// TIA Portal project "ProgettoTisc_Gruppo19" (V17)

(* hardware
DEVICE "S7-1200 station_1"  S7-1200 Station
   slot 0: "Rack_0"  S7-1200 Rack  Rack  V1.0
   slot 1: "PLC_1"  CPU 1211C DC/DC/DC  6ES7 211-1AE40-0XB0  V4.5
DEVICE "HMI_1"  KTP900 Basic PN
   slot 0: "HMI_1"  KTP900 Basic PN  6AV2 123-2JB03-0AX0  17.0.0.0
   slot 1: "HMI_RT_1"  KTP900 Basic PN  6AV2 123-2JB03-0AX0  17.0.0.0
   slot 5: "HMI_1.IE_CP_1"  PROFINET Interface  17.0.0.0
      slot 1: "PROFINET Interface_1"  PROFINET Interface
         slot 1: "Port_1"  Port
*)

// ===== PLC "PLC_1"  CPU 1211C DC/DC/DC =====

VAR_GLOBAL   // PLC tag table "Default tag table"
   "S1" AT %I10.0 : Bool;
   "Sh1" AT %I10.1 : Bool;
   "detected" AT %I10.2 : Bool;
   "X_position" AT %ID32 : Real;
   "Y_position" AT %ID36 : Real;
   "Z_position" AT %ID40 : Real;
   "S2" AT %I10.3 : Bool;
   "Sn1" AT %I10.4 : Bool;
   "S_dx" AT %I10.5 : Bool;
   "Sn_dx" AT %I10.6 : Bool;
   "Sc_value_dx" AT %ID44 : DInt;
   "exit_limit_dx" AT %I10.7 : Bool;
   "enter_limit_dx" AT %I11.0 : Bool;
   "position_dx" AT %ID48 : Real;
   "S_sx" AT %I11.1 : Bool;
   "Sn_sx" AT %I11.2 : Bool;
   "Sc_value_sx" AT %ID52 : DInt;
   "exit_limit_sx" AT %I11.3 : Bool;
   "enter_limit_sx" AT %I11.4 : Bool;
   "position_sx" AT %ID56 : Real;
   "motor1" AT %Q0.0 : Bool;
   "X_setpoint" AT %QD30 : Real;
   "Y_setpoint" AT %QD34 : Real;
   "Z_setpoint" AT %QD38 : Real;
   "grab" AT %Q0.1 : Bool;
   "motor2" AT %Q0.2 : Bool;
   "move" AT %Q0.3 : Bool;
   "move_right" AT %Q0.4 : Bool;
   "move_left" AT %Q0.5 : Bool;
   "motor_dx" AT %Q0.6 : Bool;
   "roll_dx" AT %Q0.7 : Bool;
   "motor1_dx" AT %Q1.0 : Bool;
   "motor2_dx" AT %Q1.1 : Bool;
   "motor3_dx" AT %Q1.2 : Bool;
   "setpoint_dx" AT %QD42 : Real;
   "motor_sx" AT %Q1.3 : Bool;
   "roll_sx" AT %Q1.4 : Bool;
   "motor1_sx" AT %Q1.5 : Bool;
   "motor2_sx" AT %Q1.6 : Bool;
   "motor3_sx" AT %Q1.7 : Bool;
   "setpoint_sx" AT %QD46 : Real;
   "Emitter_pallet" AT %Q2.0 : Bool;
   "Emitter_basi" AT %Q2.1 : Bool;
   "Impianto_attivo" AT %M0.0 : Bool;
   "Cmd_start" AT %M0.1 : Bool;
   "Cmd_stop" AT %M0.2 : Bool;
   "Pezzi_totali" AT %MW10 : Int;
   "Pezzi_blu" AT %MW12 : Int;
   "Pezzi_verdi" AT %MW14 : Int;
   "Pezzi_grigi" AT %MW16 : Int;
   "Allarme" AT %M0.3 : Bool;
   "Reset" AT %M0.4 : Bool;
   "Sospendi" AT %M0.5 : Bool;
   "Allarme_colore_dx" AT %M0.6 : Bool;
   "Allarme_colore_sx" AT %M0.7 : Bool;
   "Allarme_sh" AT %M1.0 : Bool;
   "Sirena_allarmi" AT %Q2.2 : Bool;
   "Flash_Sh" AT %Q2.3 : Bool;
   "Flash_dx" AT %Q2.4 : Bool;
   "Flash_sx" AT %Q2.5 : Bool;
   "Allarme_sh_int" AT %MW20 : Int;
   "Allarme_colore_dx_int" AT %MW22 : Int;
   "Allarme_colore_sx_int" AT %MW24 : Int;
   "Attesa_sh" AT %M1.1 : Bool;
   "Attesa_controllo_colore_dx" AT %M1.2 : Bool;
   "Attesa_controllo_colore_sx" AT %M1.3 : Bool;
END_VAR

DATA_BLOCK "Nastro_di_produzione_DB"   // DB1
{ S7_Optimized_Access := 'TRUE' }
VERSION : 0.1
// stored: InstanceOfName Nastro_di_produzione
"Nastro_di_produzione"
BEGIN
END_DATA_BLOCK

DATA_BLOCK "Pick-place_DB"   // DB2
{ S7_Optimized_Access := 'TRUE' }
VERSION : 0.1
// stored: InstanceOfName Pick-place
"Pick-place"
BEGIN
END_DATA_BLOCK

DATA_BLOCK "Nastro_DB"   // DB3
{ S7_Optimized_Access := 'TRUE' }
VERSION : 0.1
// stored: InstanceOfName Nastro
"Nastro"
BEGIN
END_DATA_BLOCK

DATA_BLOCK "Transfer_DB"   // DB4
{ S7_Optimized_Access := 'TRUE' }
VERSION : 0.1
// stored: InstanceOfName Transfer
"Transfer"
BEGIN
END_DATA_BLOCK

DATA_BLOCK "Nastro_di_smistamento_dx_DB"   // DB5
{ S7_Optimized_Access := 'TRUE' }
VERSION : 0.1
// stored: InstanceOfName Nastro_di_smistamento
"Nastro_di_smistamento"
BEGIN
END_DATA_BLOCK

DATA_BLOCK "Elevator_dx_DB"   // DB6
{ S7_Optimized_Access := 'TRUE' }
VERSION : 0.1
// stored: InstanceOfName Elevator
"Elevator"
BEGIN
END_DATA_BLOCK

DATA_BLOCK "Nastro_di_smistamento_sx_DB"   // DB7
{ S7_Optimized_Access := 'TRUE' }
VERSION : 0.1
// stored: InstanceOfName Nastro_di_smistamento
"Nastro_di_smistamento"
BEGIN
END_DATA_BLOCK

DATA_BLOCK "Elevator_sx_DB"   // DB8
{ S7_Optimized_Access := 'TRUE' }
VERSION : 0.1
// stored: InstanceOfName Elevator
"Elevator"
BEGIN
END_DATA_BLOCK

DATA_BLOCK "Supervisore_DB"   // DB12
{ S7_Optimized_Access := 'TRUE' }
VERSION : 0.1
// stored: InstanceOfName Supervisore
"Supervisore"
BEGIN
END_DATA_BLOCK

// folder: System blocks/Program resources

DATA_BLOCK "TON_Allarme_Sh_DB"   // DB13
{ S7_Optimized_Access := 'TRUE' }
AUTHOR : Simatic
FAMILY : IEC
NAME : IEC_TMR
VERSION : 1.0
// stored: InstanceOfName IEC_TIMER
"IEC_TIMER"
BEGIN
END_DATA_BLOCK

DATA_BLOCK "TON_Allarme_dx"   // DB14
{ S7_Optimized_Access := 'TRUE' }
AUTHOR : Simatic
FAMILY : IEC
NAME : IEC_TMR
VERSION : 1.0
// stored: InstanceOfName IEC_TIMER
"IEC_TIMER"
BEGIN
END_DATA_BLOCK

DATA_BLOCK "TON_Allarme_sx"   // DB15
{ S7_Optimized_Access := 'TRUE' }
AUTHOR : Simatic
FAMILY : IEC
NAME : IEC_TMR
VERSION : 1.0
// stored: InstanceOfName IEC_TIMER
"IEC_TIMER"
BEGIN
END_DATA_BLOCK

// folder: (top level)

FUNCTION_BLOCK "Nastro_di_produzione"   // FB1, LAD
{ S7_Optimized_Access := 'TRUE' }
VERSION : 0.1
   VAR_INPUT
      S : Bool;
      work_finished : Bool;
      Sh : Bool;
      p_dopo : Bool;
      Sospendi : Bool;
      Forza : Bool;
   END_VAR
   VAR_OUTPUT
      motor : Bool;
      work : Bool;
   END_VAR
   VAR
      p1 : Bool;
      p2 : Bool;
      p3 : Bool;
      p4 : Bool;
      p5 : Bool;
      t1 : Bool;
      t2 : Bool;
      t3 : Bool;
      t4 : Bool;
      t5 : Bool;
      R_TRIG_S : R_TRIG;
      R_TRIG_Sh : R_TRIG;
      F_TRIG_S : R_TRIG;
      INIZ : Bool;
   END_VAR
   VAR_TEMP   // added for the SCL form of the ladder/FBD networks
      _w1 : Bool;
   END_VAR
BEGIN

REGION Network 1: Inizializzazione
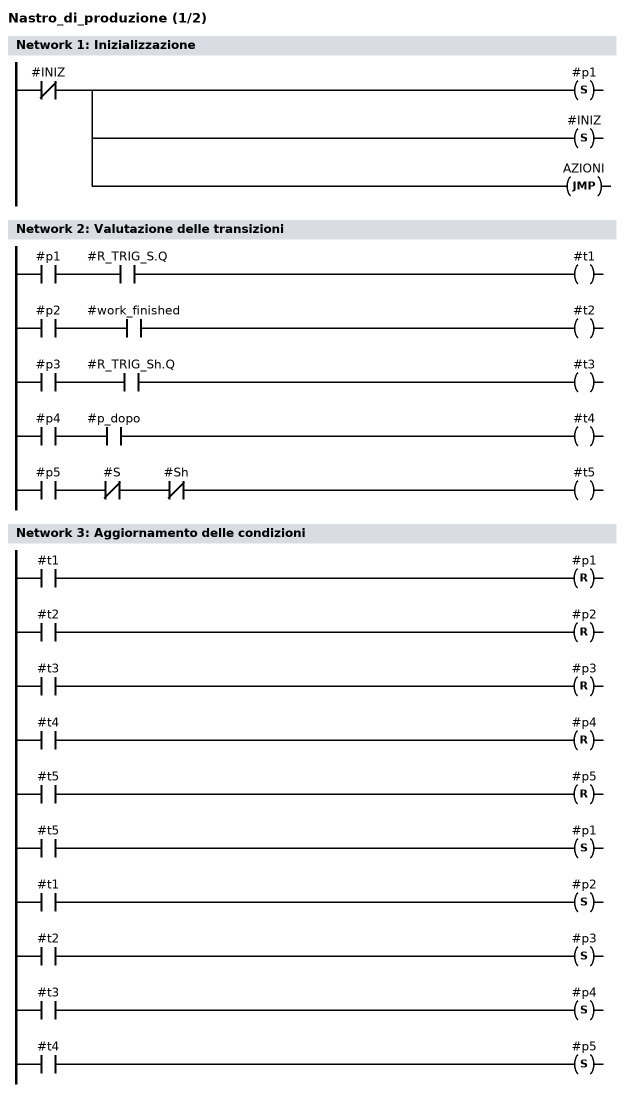
   RUNG wire#powerrail
      I_Contact( #INIZ )
      wire#w1
      S_Coil( #p1 )
   END_RUNG
   RUNG wire#w1
      S_Coil( #INIZ )
   END_RUNG
   RUNG wire#w1
      JumpCoil( AZIONI )
   END_RUNG
   // the same network as SCL:
   IF NOT #INIZ THEN #p1 := TRUE; END_IF;
   #_w1 := NOT #INIZ;
   IF #_w1 THEN
       #INIZ := TRUE;
       GOTO AZIONI;
   END_IF;
END_REGION

REGION Network 2: Valutazione delle transizioni
   RUNG wire#powerrail
      Contact( #p1 )
      Contact( #R_TRIG_S.Q )
      Coil( #t1 )
   END_RUNG
   RUNG wire#powerrail
      Contact( #p2 )
      Contact( #work_finished )
      Coil( #t2 )
   END_RUNG
   RUNG wire#powerrail
      Contact( #p3 )
      Contact( #R_TRIG_Sh.Q )
      Coil( #t3 )
   END_RUNG
   RUNG wire#powerrail
      Contact( #p4 )
      Contact( #p_dopo )
      Coil( #t4 )
   END_RUNG
   RUNG wire#powerrail
      Contact( #p5 )
      I_Contact( #S )
      I_Contact( #Sh )
      Coil( #t5 )
   END_RUNG
   // the same network as SCL:
   #t1 := #p1 AND #R_TRIG_S.Q;
   #t2 := #p2 AND #work_finished;
   #t3 := #p3 AND #R_TRIG_Sh.Q;
   #t4 := #p4 AND #p_dopo;
   #t5 := #p5 AND NOT #S AND NOT #Sh;
END_REGION

REGION Network 3: Aggiornamento delle condizioni
   RUNG wire#powerrail
      Contact( #t1 )
      R_Coil( #p1 )
   END_RUNG
   RUNG wire#powerrail
      Contact( #t2 )
      R_Coil( #p2 )
   END_RUNG
   RUNG wire#powerrail
      Contact( #t3 )
      R_Coil( #p3 )
   END_RUNG
   RUNG wire#powerrail
      Contact( #t4 )
      R_Coil( #p4 )
   END_RUNG
   RUNG wire#powerrail
      Contact( #t5 )
      R_Coil( #p5 )
   END_RUNG
   RUNG wire#powerrail
      Contact( #t5 )
      S_Coil( #p1 )
   END_RUNG
   RUNG wire#powerrail
      Contact( #t1 )
      S_Coil( #p2 )
   END_RUNG
   RUNG wire#powerrail
      Contact( #t2 )
      S_Coil( #p3 )
   END_RUNG
   RUNG wire#powerrail
      Contact( #t3 )
      S_Coil( #p4 )
   END_RUNG
   RUNG wire#powerrail
      Contact( #t4 )
      S_Coil( #p5 )
   END_RUNG
   // the same network as SCL:
   IF #t1 THEN #p1 := FALSE; END_IF;
   IF #t2 THEN #p2 := FALSE; END_IF;
   IF #t3 THEN #p3 := FALSE; END_IF;
   IF #t4 THEN #p4 := FALSE; END_IF;
   IF #t5 THEN
       #p5 := FALSE;
       #p1 := TRUE;
   END_IF;
   IF #t1 THEN #p2 := TRUE; END_IF;
   IF #t2 THEN #p3 := TRUE; END_IF;
   IF #t3 THEN #p4 := TRUE; END_IF;
   IF #t4 THEN #p5 := TRUE; END_IF;
END_REGION

REGION Network 4: Macroazioni di sospensione e forzatura alla fase 1 e sezione di esecuzione delle azioni
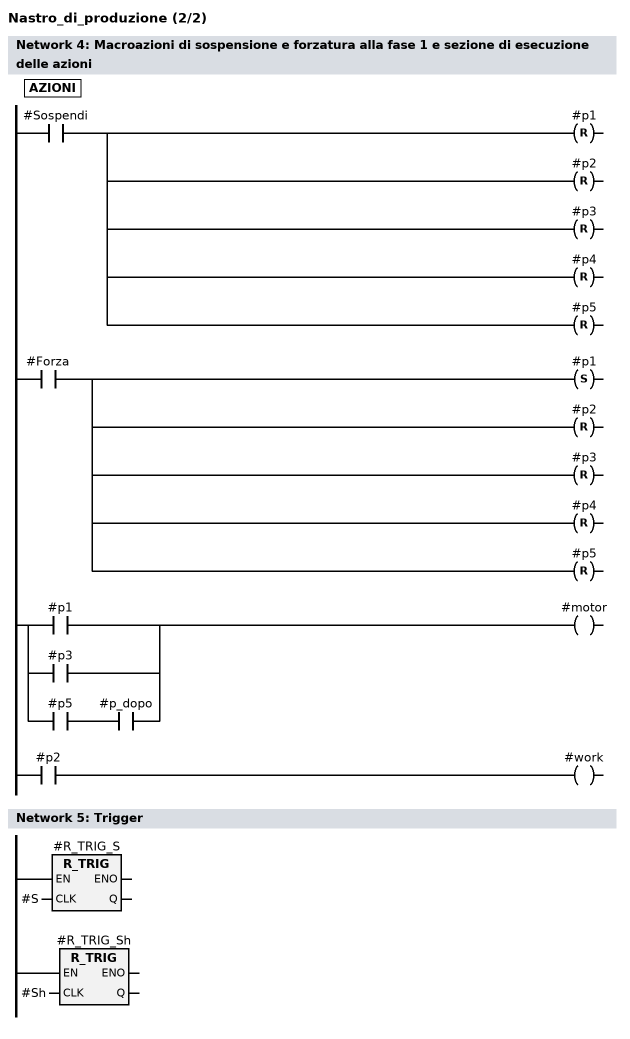
   Label( AZIONI )
   RUNG wire#powerrail
      Contact( #Sospendi )
      wire#w1
      R_Coil( #p1 )
   END_RUNG
   RUNG wire#w1
      R_Coil( #p2 )
   END_RUNG
   RUNG wire#w1
      R_Coil( #p3 )
   END_RUNG
   RUNG wire#w1
      R_Coil( #p4 )
   END_RUNG
   RUNG wire#w1
      R_Coil( #p5 )
   END_RUNG
   RUNG wire#powerrail
      Contact( #Forza )
      wire#w2
      S_Coil( #p1 )
   END_RUNG
   RUNG wire#w2
      R_Coil( #p2 )
   END_RUNG
   RUNG wire#w2
      R_Coil( #p3 )
   END_RUNG
   RUNG wire#w2
      R_Coil( #p4 )
   END_RUNG
   RUNG wire#w2
      R_Coil( #p5 )
   END_RUNG
   RUNG wire#powerrail
      Contact( #p1 )
      wire#w3
      Coil( #motor )
   END_RUNG
   RUNG wire#powerrail
      Contact( #p3 )
   END_RUNG wire#w3
   RUNG wire#powerrail
      Contact( #p5 )
      Contact( #p_dopo )
   END_RUNG wire#w3
   RUNG wire#powerrail
      Contact( #p2 )
      Coil( #work )
   END_RUNG
   // the same network as SCL:
   AZIONI:
   IF #Sospendi THEN
       #p1 := FALSE;
       #p2 := FALSE;
       #p3 := FALSE;
       #p4 := FALSE;
       #p5 := FALSE;
   END_IF;
   IF #Forza THEN
       #p1 := TRUE;
       #p2 := FALSE;
       #p3 := FALSE;
       #p4 := FALSE;
       #p5 := FALSE;
   END_IF;
   #motor := #p1 OR #p3 OR (#p5 AND #p_dopo);
   #work := #p2;
END_REGION

REGION Network 5: Trigger
   #R_TRIG_S(CLK := #S);   // R_TRIG
   #R_TRIG_Sh(CLK := #Sh);   // R_TRIG
END_REGION
END_FUNCTION_BLOCK

FUNCTION_BLOCK "Nastro"   // FB2, LAD
{ S7_Optimized_Access := 'TRUE' }
VERSION : 0.1
   VAR_INPUT
      S : Bool;
      p_dopo : Bool;
      Sospendi : Bool;
      Forza : Bool;
   END_VAR
   VAR_OUTPUT
      Motor : Bool;
      Pronto_ricevere : Bool;
      transfer : Bool;
   END_VAR
   VAR
      p1 : Bool;
      p2 : Bool;
      p3 : Bool;
      t1 : Bool;
      t2 : Bool;
      t3 : Bool;
      R_TRIG_S : R_TRIG;
      F_TRIG_S : F_TRIG;
      INIZ : Bool;
   END_VAR
   VAR_TEMP   // added for the SCL form of the ladder/FBD networks
      _w1 : Bool;
   END_VAR
BEGIN

REGION Network 1: Inizializzazione
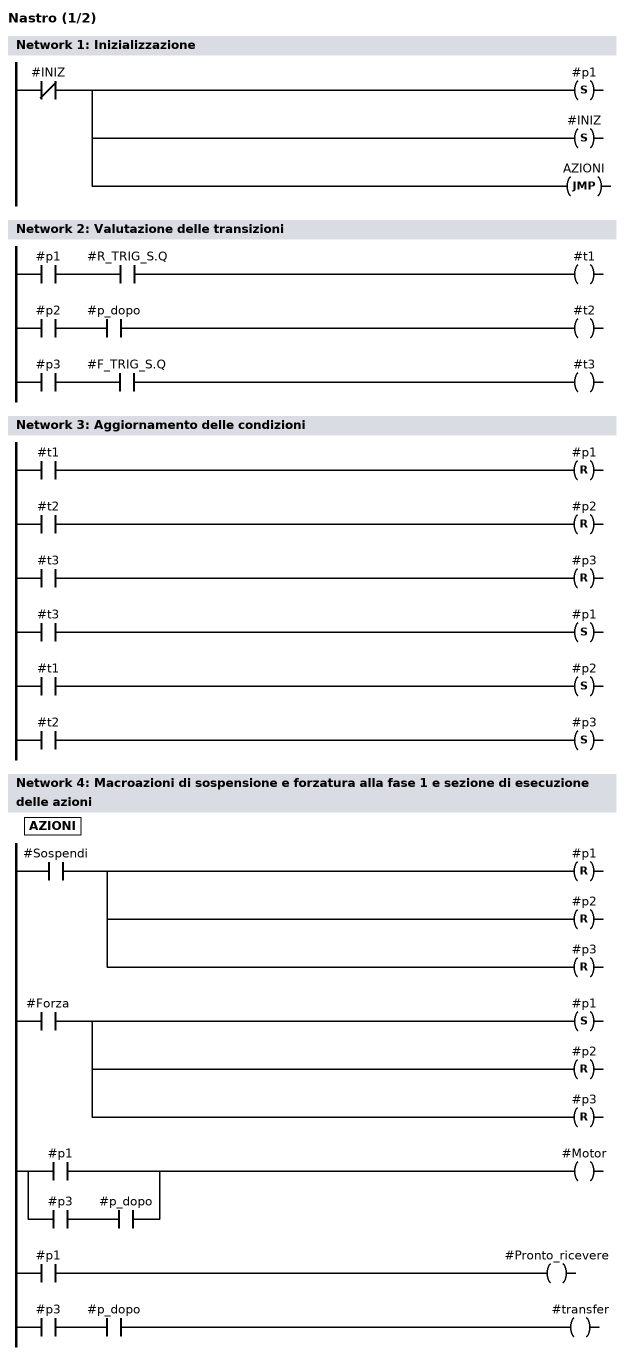
   RUNG wire#powerrail
      I_Contact( #INIZ )
      wire#w1
      S_Coil( #p1 )
   END_RUNG
   RUNG wire#w1
      S_Coil( #INIZ )
   END_RUNG
   RUNG wire#w1
      JumpCoil( AZIONI )
   END_RUNG
   // the same network as SCL:
   IF NOT #INIZ THEN #p1 := TRUE; END_IF;
   #_w1 := NOT #INIZ;
   IF #_w1 THEN
       #INIZ := TRUE;
       GOTO AZIONI;
   END_IF;
END_REGION

REGION Network 2: Valutazione delle transizioni
   RUNG wire#powerrail
      Contact( #p1 )
      Contact( #R_TRIG_S.Q )
      Coil( #t1 )
   END_RUNG
   RUNG wire#powerrail
      Contact( #p2 )
      Contact( #p_dopo )
      Coil( #t2 )
   END_RUNG
   RUNG wire#powerrail
      Contact( #p3 )
      Contact( #F_TRIG_S.Q )
      Coil( #t3 )
   END_RUNG
   // the same network as SCL:
   #t1 := #p1 AND #R_TRIG_S.Q;
   #t2 := #p2 AND #p_dopo;
   #t3 := #p3 AND #F_TRIG_S.Q;
END_REGION

REGION Network 3: Aggiornamento delle condizioni
   RUNG wire#powerrail
      Contact( #t1 )
      R_Coil( #p1 )
   END_RUNG
   RUNG wire#powerrail
      Contact( #t2 )
      R_Coil( #p2 )
   END_RUNG
   RUNG wire#powerrail
      Contact( #t3 )
      R_Coil( #p3 )
   END_RUNG
   RUNG wire#powerrail
      Contact( #t3 )
      S_Coil( #p1 )
   END_RUNG
   RUNG wire#powerrail
      Contact( #t1 )
      S_Coil( #p2 )
   END_RUNG
   RUNG wire#powerrail
      Contact( #t2 )
      S_Coil( #p3 )
   END_RUNG
   // the same network as SCL:
   IF #t1 THEN #p1 := FALSE; END_IF;
   IF #t2 THEN #p2 := FALSE; END_IF;
   IF #t3 THEN
       #p3 := FALSE;
       #p1 := TRUE;
   END_IF;
   IF #t1 THEN #p2 := TRUE; END_IF;
   IF #t2 THEN #p3 := TRUE; END_IF;
END_REGION

REGION Network 4: Macroazioni di sospensione e forzatura alla fase 1 e sezione di esecuzione delle azioni
   Label( AZIONI )
   RUNG wire#powerrail
      Contact( #Sospendi )
      wire#w1
      R_Coil( #p1 )
   END_RUNG
   RUNG wire#w1
      R_Coil( #p2 )
   END_RUNG
   RUNG wire#w1
      R_Coil( #p3 )
   END_RUNG
   RUNG wire#powerrail
      Contact( #Forza )
      wire#w2
      S_Coil( #p1 )
   END_RUNG
   RUNG wire#w2
      R_Coil( #p2 )
   END_RUNG
   RUNG wire#w2
      R_Coil( #p3 )
   END_RUNG
   RUNG wire#powerrail
      Contact( #p1 )
      wire#w3
      Coil( #Motor )
   END_RUNG
   RUNG wire#powerrail
      Contact( #p3 )
      Contact( #p_dopo )
   END_RUNG wire#w3
   RUNG wire#powerrail
      Contact( #p1 )
      Coil( #Pronto_ricevere )
   END_RUNG
   RUNG wire#powerrail
      Contact( #p3 )
      Contact( #p_dopo )
      Coil( #transfer )
   END_RUNG
   // the same network as SCL:
   AZIONI:
   IF #Sospendi THEN
       #p1 := FALSE;
       #p2 := FALSE;
       #p3 := FALSE;
   END_IF;
   IF #Forza THEN
       #p1 := TRUE;
       #p2 := FALSE;
       #p3 := FALSE;
   END_IF;
   #Motor := #p1 OR (#p3 AND #p_dopo);
   #Pronto_ricevere := #p1;
   #transfer := #p3 AND #p_dopo;
END_REGION

REGION Network 5: Trigger
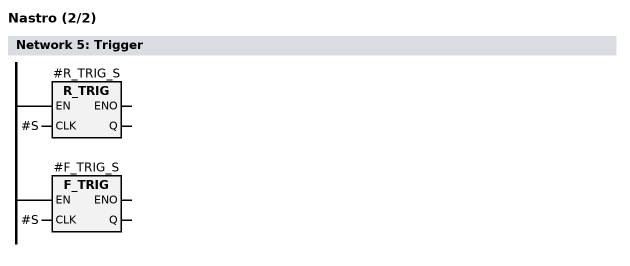
   #R_TRIG_S(CLK := #S);   // R_TRIG
   #F_TRIG_S(CLK := #S);   // F_TRIG
END_REGION
END_FUNCTION_BLOCK

FUNCTION_BLOCK "Supervisore"   // FB3, LAD
{ S7_Optimized_Access := 'TRUE' }
VERSION : 0.1
   VAR_INPUT
      Sospendi : Bool;
      Reset : Bool;
      Allarme : Bool;
   END_VAR
   VAR_OUTPUT
      Cmd_Sospendi : Bool;
      Cmd_Forzatura : Bool;
      Stato_sospeso : Bool;
   END_VAR
   VAR
      p1 : Bool;
      p2 : Bool;
      p3 : Bool;
      p4 : Bool;
      t1 : Bool;
      t2 : Bool;
      t3 : Bool;
      t4 : Bool;
      INIZ : Bool;
   END_VAR
   VAR_TEMP   // added for the SCL form of the ladder/FBD networks
      _w1 : Bool;
   END_VAR
BEGIN

REGION Network 1: Inizializzazione
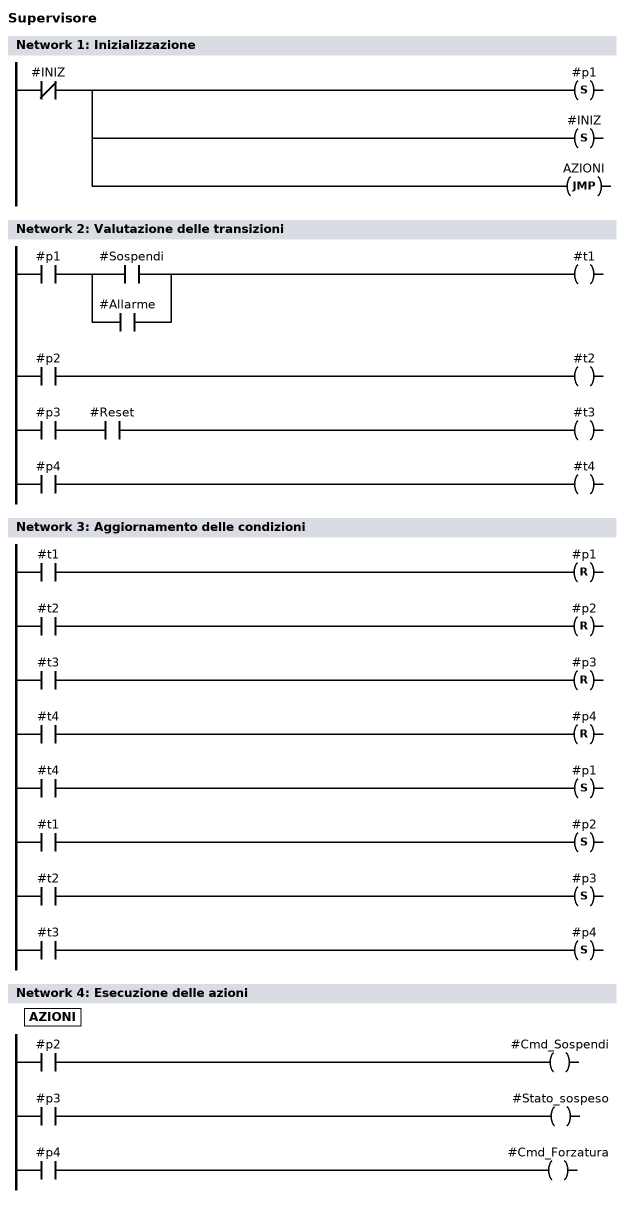
   RUNG wire#powerrail
      I_Contact( #INIZ )
      wire#w1
      S_Coil( #p1 )
   END_RUNG
   RUNG wire#w1
      S_Coil( #INIZ )
   END_RUNG
   RUNG wire#w1
      JumpCoil( AZIONI )
   END_RUNG
   // the same network as SCL:
   IF NOT #INIZ THEN #p1 := TRUE; END_IF;
   #_w1 := NOT #INIZ;
   IF #_w1 THEN
       #INIZ := TRUE;
       GOTO AZIONI;
   END_IF;
END_REGION

REGION Network 2: Valutazione delle transizioni
   RUNG wire#powerrail
      Contact( #p1 )
      wire#w1
      Contact( #Sospendi )
      wire#w2
      Coil( #t1 )
   END_RUNG
   RUNG wire#w1
      Contact( #Allarme )
   END_RUNG wire#w2
   RUNG wire#powerrail
      Contact( #p2 )
      Coil( #t2 )
   END_RUNG
   RUNG wire#powerrail
      Contact( #p3 )
      Contact( #Reset )
      Coil( #t3 )
   END_RUNG
   RUNG wire#powerrail
      Contact( #p4 )
      Coil( #t4 )
   END_RUNG
   // the same network as SCL:
   #t1 := #p1 AND (#Sospendi OR #Allarme);
   #t2 := #p2;
   #t3 := #p3 AND #Reset;
   #t4 := #p4;
END_REGION

REGION Network 3: Aggiornamento delle condizioni
   RUNG wire#powerrail
      Contact( #t1 )
      R_Coil( #p1 )
   END_RUNG
   RUNG wire#powerrail
      Contact( #t2 )
      R_Coil( #p2 )
   END_RUNG
   RUNG wire#powerrail
      Contact( #t3 )
      R_Coil( #p3 )
   END_RUNG
   RUNG wire#powerrail
      Contact( #t4 )
      R_Coil( #p4 )
   END_RUNG
   RUNG wire#powerrail
      Contact( #t4 )
      S_Coil( #p1 )
   END_RUNG
   RUNG wire#powerrail
      Contact( #t1 )
      S_Coil( #p2 )
   END_RUNG
   RUNG wire#powerrail
      Contact( #t2 )
      S_Coil( #p3 )
   END_RUNG
   RUNG wire#powerrail
      Contact( #t3 )
      S_Coil( #p4 )
   END_RUNG
   // the same network as SCL:
   IF #t1 THEN #p1 := FALSE; END_IF;
   IF #t2 THEN #p2 := FALSE; END_IF;
   IF #t3 THEN #p3 := FALSE; END_IF;
   IF #t4 THEN
       #p4 := FALSE;
       #p1 := TRUE;
   END_IF;
   IF #t1 THEN #p2 := TRUE; END_IF;
   IF #t2 THEN #p3 := TRUE; END_IF;
   IF #t3 THEN #p4 := TRUE; END_IF;
END_REGION

REGION Network 4: Esecuzione delle azioni
   Label( AZIONI )
   RUNG wire#powerrail
      Contact( #p2 )
      Coil( #Cmd_Sospendi )
   END_RUNG
   RUNG wire#powerrail
      Contact( #p3 )
      Coil( #Stato_sospeso )
   END_RUNG
   RUNG wire#powerrail
      Contact( #p4 )
      Coil( #Cmd_Forzatura )
   END_RUNG
   // the same network as SCL:
   AZIONI:
   #Cmd_Sospendi := #p2;
   #Stato_sospeso := #p3;
   #Cmd_Forzatura := #p4;
END_REGION
END_FUNCTION_BLOCK

FUNCTION_BLOCK "Transfer"   // FB4, LAD
{ S7_Optimized_Access := 'TRUE' }
VERSION : 0.1
   VAR_INPUT
      Sn : Bool;
      transfer : Bool;
      p_dopo_dx : Bool;
      p_dopo_sx : Bool;
      transfer_finished_dx : Bool;
      transfer_finished_sx : Bool;
      Sospendi : Bool;
      Forza : Bool;
   END_VAR
   VAR_OUTPUT
      Pronto_ricevere : Bool;
      Move : Bool;
      Move_right : Bool;
      Move_left : Bool;
   END_VAR
   VAR
      p1 : Bool;
      p2 : Bool;
      p3 : Bool;
      p4 : Bool;
      p5 : Bool;
      t1 : Bool;
      t2 : Bool;
      t3 : Bool;
      t4 : Bool;
      t5 : Bool;
      t6 : Bool;
      INIZ : Bool;
      R_TRIG_Transfer : R_TRIG;
      R_TRIG_Sn : R_TRIG;
      Timer_f2 : TON_TIME;
   END_VAR
   VAR_TEMP   // added for the SCL form of the ladder/FBD networks
      _w1 : Bool;
   END_VAR
BEGIN

REGION Network 1: Inizializzazione
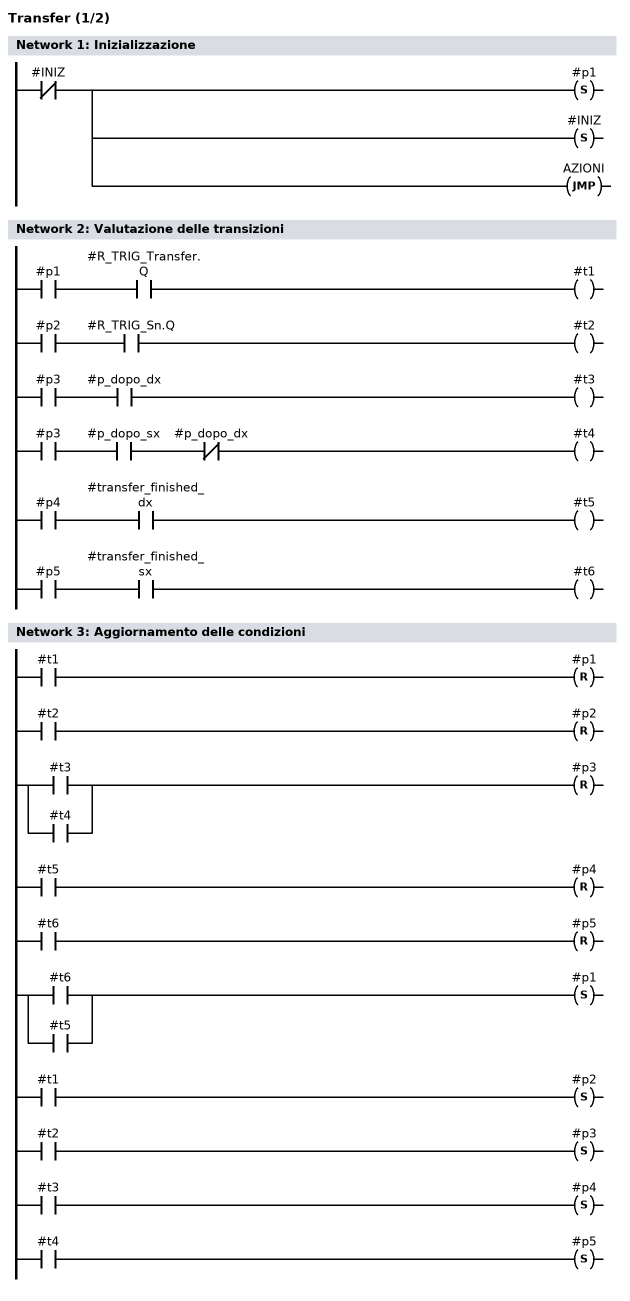
   RUNG wire#powerrail
      I_Contact( #INIZ )
      wire#w1
      S_Coil( #p1 )
   END_RUNG
   RUNG wire#w1
      S_Coil( #INIZ )
   END_RUNG
   RUNG wire#w1
      JumpCoil( AZIONI )
   END_RUNG
   // the same network as SCL:
   IF NOT #INIZ THEN #p1 := TRUE; END_IF;
   #_w1 := NOT #INIZ;
   IF #_w1 THEN
       #INIZ := TRUE;
       GOTO AZIONI;
   END_IF;
END_REGION

REGION Network 2: Valutazione delle transizioni
   RUNG wire#powerrail
      Contact( #p1 )
      Contact( #R_TRIG_Transfer.Q )
      Coil( #t1 )
   END_RUNG
   RUNG wire#powerrail
      Contact( #p2 )
      Contact( #R_TRIG_Sn.Q )
      Coil( #t2 )
   END_RUNG
   RUNG wire#powerrail
      Contact( #p3 )
      Contact( #p_dopo_dx )
      Coil( #t3 )
   END_RUNG
   RUNG wire#powerrail
      Contact( #p3 )
      Contact( #p_dopo_sx )
      I_Contact( #p_dopo_dx )
      Coil( #t4 )
   END_RUNG
   RUNG wire#powerrail
      Contact( #p4 )
      Contact( #transfer_finished_dx )
      Coil( #t5 )
   END_RUNG
   RUNG wire#powerrail
      Contact( #p5 )
      Contact( #transfer_finished_sx )
      Coil( #t6 )
   END_RUNG
   // the same network as SCL:
   #t1 := #p1 AND #R_TRIG_Transfer.Q;
   #t2 := #p2 AND #R_TRIG_Sn.Q;
   #t3 := #p3 AND #p_dopo_dx;
   #t4 := #p3 AND #p_dopo_sx AND NOT #p_dopo_dx;
   #t5 := #p4 AND #transfer_finished_dx;
   #t6 := #p5 AND #transfer_finished_sx;
END_REGION

REGION Network 3: Aggiornamento delle condizioni
   RUNG wire#powerrail
      Contact( #t1 )
      R_Coil( #p1 )
   END_RUNG
   RUNG wire#powerrail
      Contact( #t2 )
      R_Coil( #p2 )
   END_RUNG
   RUNG wire#powerrail
      Contact( #t3 )
      wire#w1
      R_Coil( #p3 )
   END_RUNG
   RUNG wire#powerrail
      Contact( #t4 )
   END_RUNG wire#w1
   RUNG wire#powerrail
      Contact( #t5 )
      R_Coil( #p4 )
   END_RUNG
   RUNG wire#powerrail
      Contact( #t6 )
      R_Coil( #p5 )
   END_RUNG
   RUNG wire#powerrail
      Contact( #t6 )
      wire#w2
      S_Coil( #p1 )
   END_RUNG
   RUNG wire#powerrail
      Contact( #t5 )
   END_RUNG wire#w2
   RUNG wire#powerrail
      Contact( #t1 )
      S_Coil( #p2 )
   END_RUNG
   RUNG wire#powerrail
      Contact( #t2 )
      S_Coil( #p3 )
   END_RUNG
   RUNG wire#powerrail
      Contact( #t3 )
      S_Coil( #p4 )
   END_RUNG
   RUNG wire#powerrail
      Contact( #t4 )
      S_Coil( #p5 )
   END_RUNG
   // the same network as SCL:
   IF #t1 THEN #p1 := FALSE; END_IF;
   IF #t2 THEN #p2 := FALSE; END_IF;
   IF #t3 OR #t4 THEN #p3 := FALSE; END_IF;
   IF #t5 THEN #p4 := FALSE; END_IF;
   IF #t6 THEN #p5 := FALSE; END_IF;
   IF #t6 OR #t5 THEN #p1 := TRUE; END_IF;
   IF #t1 THEN #p2 := TRUE; END_IF;
   IF #t2 THEN #p3 := TRUE; END_IF;
   IF #t3 THEN #p4 := TRUE; END_IF;
   IF #t4 THEN #p5 := TRUE; END_IF;
END_REGION

REGION Network 4: Macroazioni di sospensione e forzatura alla fase 1 e sezione di esecuzione delle azioni
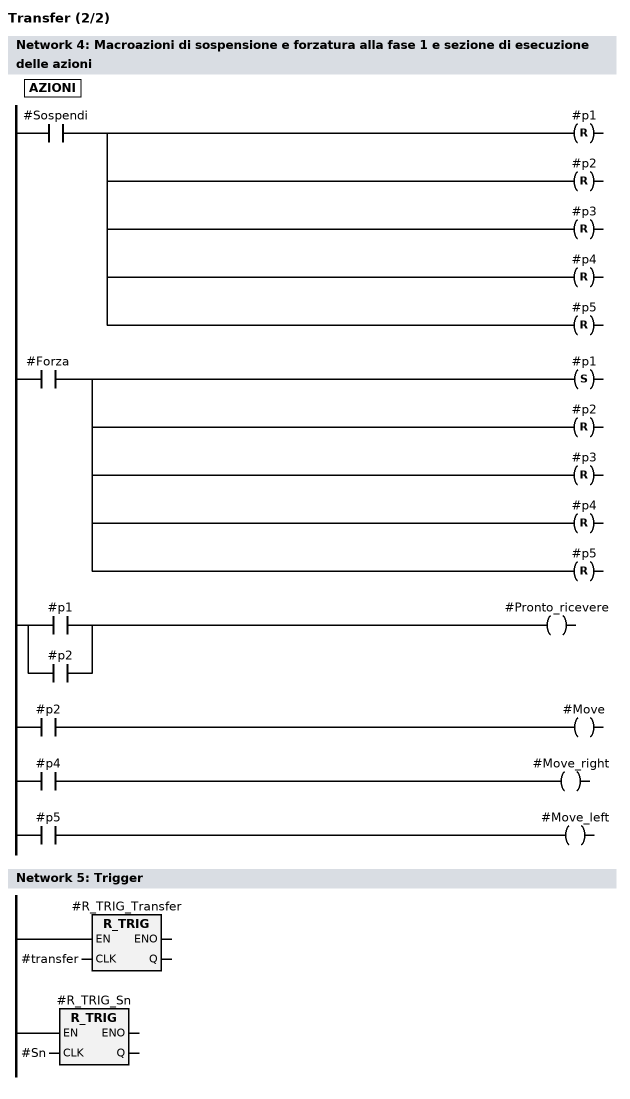
   Label( AZIONI )
   RUNG wire#powerrail
      Contact( #Sospendi )
      wire#w1
      R_Coil( #p1 )
   END_RUNG
   RUNG wire#w1
      R_Coil( #p2 )
   END_RUNG
   RUNG wire#w1
      R_Coil( #p3 )
   END_RUNG
   RUNG wire#w1
      R_Coil( #p4 )
   END_RUNG
   RUNG wire#w1
      R_Coil( #p5 )
   END_RUNG
   RUNG wire#powerrail
      Contact( #Forza )
      wire#w2
      S_Coil( #p1 )
   END_RUNG
   RUNG wire#w2
      R_Coil( #p2 )
   END_RUNG
   RUNG wire#w2
      R_Coil( #p3 )
   END_RUNG
   RUNG wire#w2
      R_Coil( #p4 )
   END_RUNG
   RUNG wire#w2
      R_Coil( #p5 )
   END_RUNG
   RUNG wire#powerrail
      Contact( #p1 )
      wire#w3
      Coil( #Pronto_ricevere )
   END_RUNG
   RUNG wire#powerrail
      Contact( #p2 )
   END_RUNG wire#w3
   RUNG wire#powerrail
      Contact( #p2 )
      Coil( #Move )
   END_RUNG
   RUNG wire#powerrail
      Contact( #p4 )
      Coil( #Move_right )
   END_RUNG
   RUNG wire#powerrail
      Contact( #p5 )
      Coil( #Move_left )
   END_RUNG
   // the same network as SCL:
   AZIONI:
   IF #Sospendi THEN
       #p1 := FALSE;
       #p2 := FALSE;
       #p3 := FALSE;
       #p4 := FALSE;
       #p5 := FALSE;
   END_IF;
   IF #Forza THEN
       #p1 := TRUE;
       #p2 := FALSE;
       #p3 := FALSE;
       #p4 := FALSE;
       #p5 := FALSE;
   END_IF;
   #Pronto_ricevere := #p1 OR #p2;
   #Move := #p2;
   #Move_right := #p4;
   #Move_left := #p5;
END_REGION

REGION Network 5: Trigger
   #R_TRIG_Transfer(CLK := #transfer);   // R_TRIG
   #R_TRIG_Sn(CLK := #Sn);   // R_TRIG
END_REGION
END_FUNCTION_BLOCK

FUNCTION_BLOCK "Nastro_di_smistamento"   // FB5, LAD
{ S7_Optimized_Access := 'TRUE' }
VERSION : 0.1
   VAR_INPUT
      S : Bool;
      Sn : Bool;
      Sc_value : Int;
      p_dopo : Bool;
      Sospendi : Bool;
      Forza : Bool;
   END_VAR
   VAR_OUTPUT
      Motor : Bool;
      pronto_ricevere : Bool;
      transfer_finished : Bool;
      piano_elevator : Int;
   END_VAR
   VAR
      p1 : Bool;
      p2 : Bool;
      p3 : Bool;
      p4 : Bool;
      p5 : Bool;
      p6 : Bool;
      p7 : Bool;
      t1 : Bool;
      t2 : Bool;
      t3 : Bool;
      t4 : Bool;
      t5 : Bool;
      t6 : Bool;
      t7 : Bool;
      INIZ : Bool;
      Colore_mem : Int;
      R_TRIG_S : R_TRIG;
      R_TRIG_SN : R_TRIG;
      timer_p2 : TON_TIME;
      timer_p4 : TON_TIME;
   END_VAR
   VAR_TEMP   // added for the SCL form of the ladder/FBD networks
      _w1 : Bool;
   END_VAR
BEGIN

REGION Network 1: Inizializzazione
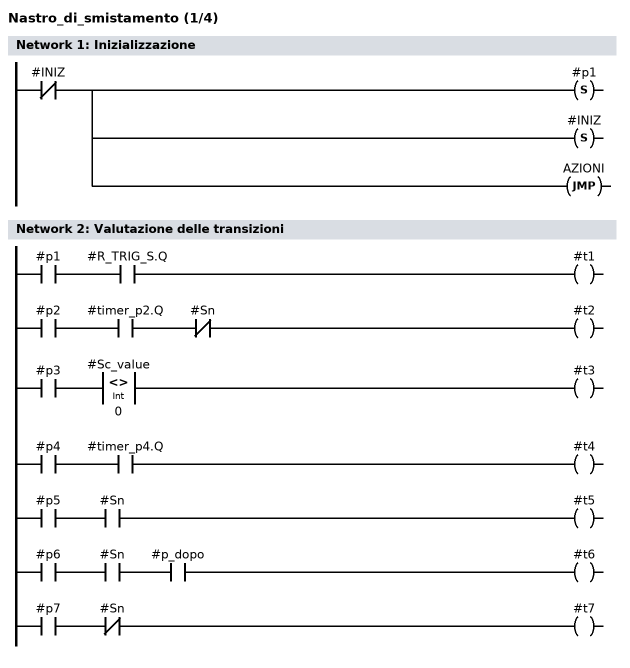
   RUNG wire#powerrail
      I_Contact( #INIZ )
      wire#w1
      S_Coil( #p1 )
   END_RUNG
   RUNG wire#w1
      S_Coil( #INIZ )
   END_RUNG
   RUNG wire#w1
      JumpCoil( AZIONI )
   END_RUNG
   // the same network as SCL:
   IF NOT #INIZ THEN #p1 := TRUE; END_IF;
   #_w1 := NOT #INIZ;
   IF #_w1 THEN
       #INIZ := TRUE;
       GOTO AZIONI;
   END_IF;
END_REGION

REGION Network 2: Valutazione delle transizioni
   RUNG wire#powerrail
      Contact( #p1 )
      Contact( #R_TRIG_S.Q )
      Coil( #t1 )
   END_RUNG
   RUNG wire#powerrail
      Contact( #p2 )
      Contact( #timer_p2.Q )
      I_Contact( #Sn )
      Coil( #t2 )
   END_RUNG
   RUNG wire#powerrail
      Contact( #p3 )
      { S7_Templates := "SrcType := Int" } NE_Contact(in1 := #Sc_value, in2 := 0)
      Coil( #t3 )
   END_RUNG
   RUNG wire#powerrail
      Contact( #p4 )
      Contact( #timer_p4.Q )
      Coil( #t4 )
   END_RUNG
   RUNG wire#powerrail
      Contact( #p5 )
      Contact( #Sn )
      Coil( #t5 )
   END_RUNG
   RUNG wire#powerrail
      Contact( #p6 )
      Contact( #Sn )
      Contact( #p_dopo )
      Coil( #t6 )
   END_RUNG
   RUNG wire#powerrail
      Contact( #p7 )
      I_Contact( #Sn )
      Coil( #t7 )
   END_RUNG
   // the same network as SCL:
   #t1 := #p1 AND #R_TRIG_S.Q;
   #t2 := #p2 AND #timer_p2.Q AND NOT #Sn;
   #t3 := #p3 AND (#Sc_value <> 0);
   #t4 := #p4 AND #timer_p4.Q;
   #t5 := #p5 AND #Sn;
   #t6 := #p6 AND #Sn AND #p_dopo;
   #t7 := #p7 AND NOT #Sn;
END_REGION

REGION Network 3: Aggiornamento delle condizioni
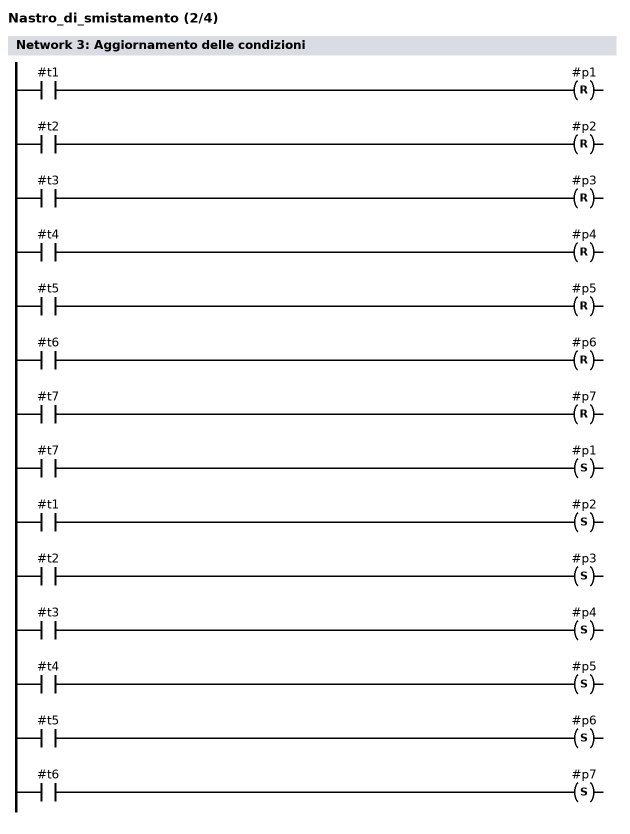
   RUNG wire#powerrail
      Contact( #t1 )
      R_Coil( #p1 )
   END_RUNG
   RUNG wire#powerrail
      Contact( #t2 )
      R_Coil( #p2 )
   END_RUNG
   RUNG wire#powerrail
      Contact( #t3 )
      R_Coil( #p3 )
   END_RUNG
   RUNG wire#powerrail
      Contact( #t4 )
      R_Coil( #p4 )
   END_RUNG
   RUNG wire#powerrail
      Contact( #t5 )
      R_Coil( #p5 )
   END_RUNG
   RUNG wire#powerrail
      Contact( #t6 )
      R_Coil( #p6 )
   END_RUNG
   RUNG wire#powerrail
      Contact( #t7 )
      R_Coil( #p7 )
   END_RUNG
   RUNG wire#powerrail
      Contact( #t7 )
      S_Coil( #p1 )
   END_RUNG
   RUNG wire#powerrail
      Contact( #t1 )
      S_Coil( #p2 )
   END_RUNG
   RUNG wire#powerrail
      Contact( #t2 )
      S_Coil( #p3 )
   END_RUNG
   RUNG wire#powerrail
      Contact( #t3 )
      S_Coil( #p4 )
   END_RUNG
   RUNG wire#powerrail
      Contact( #t4 )
      S_Coil( #p5 )
   END_RUNG
   RUNG wire#powerrail
      Contact( #t5 )
      S_Coil( #p6 )
   END_RUNG
   RUNG wire#powerrail
      Contact( #t6 )
      S_Coil( #p7 )
   END_RUNG
   // the same network as SCL:
   IF #t1 THEN #p1 := FALSE; END_IF;
   IF #t2 THEN #p2 := FALSE; END_IF;
   IF #t3 THEN #p3 := FALSE; END_IF;
   IF #t4 THEN #p4 := FALSE; END_IF;
   IF #t5 THEN #p5 := FALSE; END_IF;
   IF #t6 THEN #p6 := FALSE; END_IF;
   IF #t7 THEN
       #p7 := FALSE;
       #p1 := TRUE;
   END_IF;
   IF #t1 THEN #p2 := TRUE; END_IF;
   IF #t2 THEN #p3 := TRUE; END_IF;
   IF #t3 THEN #p4 := TRUE; END_IF;
   IF #t4 THEN #p5 := TRUE; END_IF;
   IF #t5 THEN #p6 := TRUE; END_IF;
   IF #t6 THEN #p7 := TRUE; END_IF;
END_REGION

REGION Network 4: Macroazioni di sospensione e forzatura alla fase 1 e sezione di esecuzione delle azioni
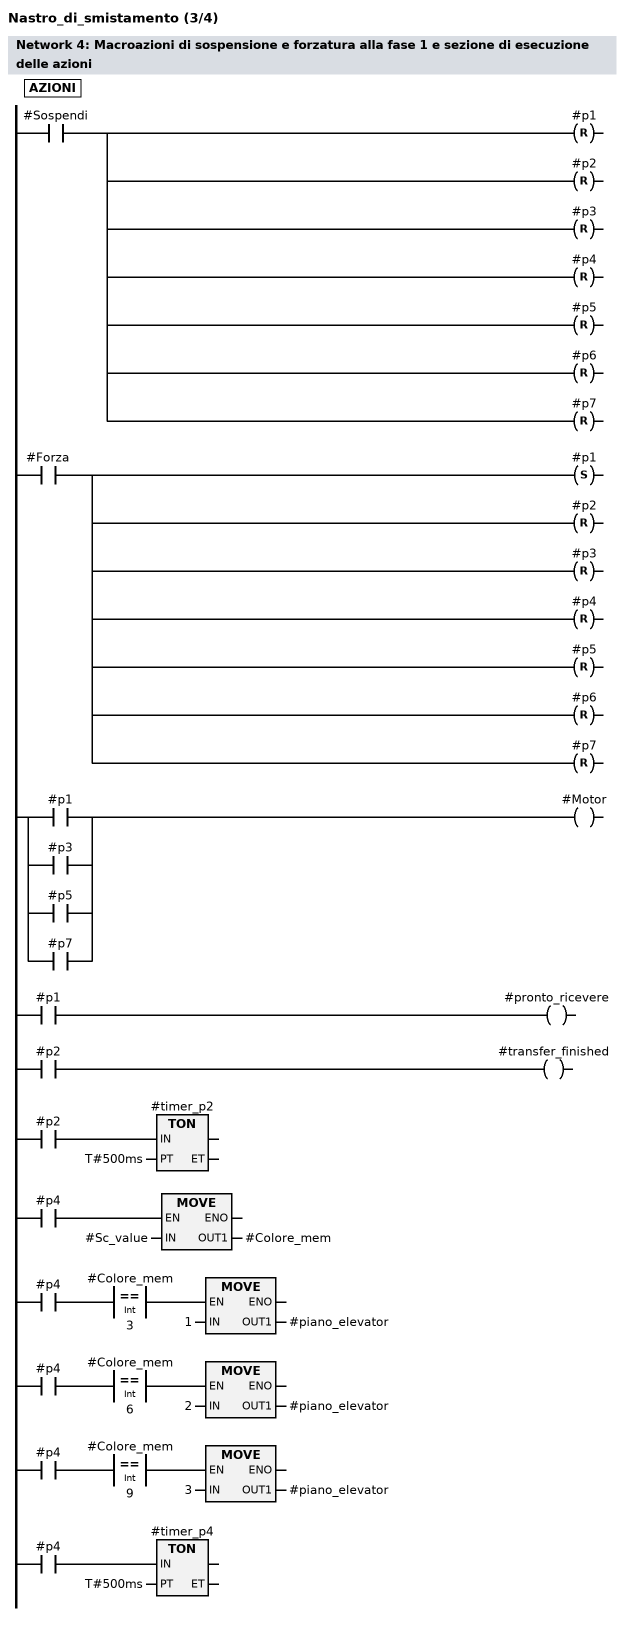
   AZIONI:
   IF #Sospendi THEN
       #p1 := FALSE;
       #p2 := FALSE;
       #p3 := FALSE;
       #p4 := FALSE;
       #p5 := FALSE;
       #p6 := FALSE;
       #p7 := FALSE;
   END_IF;
   IF #Forza THEN
       #p1 := TRUE;
       #p2 := FALSE;
       #p3 := FALSE;
       #p4 := FALSE;
       #p5 := FALSE;
       #p6 := FALSE;
       #p7 := FALSE;
   END_IF;
   #Motor := #p1 OR #p3 OR #p5 OR #p7;
   #pronto_ricevere := #p1;
   #transfer_finished := #p2;
   #timer_p2(IN := #p2, PT := T#500ms);   // TON
   IF #p4 THEN #Colore_mem := #Sc_value; END_IF;
   IF #p4 AND (#Colore_mem = 3) THEN #piano_elevator := 1; END_IF;
   IF #p4 AND (#Colore_mem = 6) THEN #piano_elevator := 2; END_IF;
   IF #p4 AND (#Colore_mem = 9) THEN #piano_elevator := 3; END_IF;
   #timer_p4(IN := #p4, PT := T#500ms);   // TON
END_REGION

REGION Network 5: Trigger
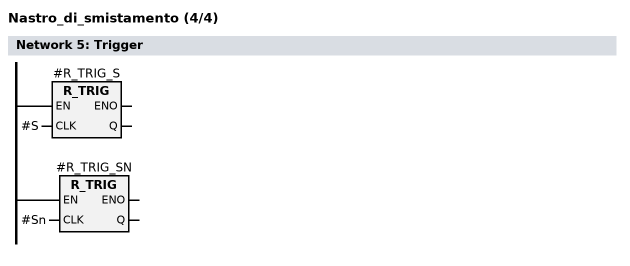
   #R_TRIG_S(CLK := #S);   // R_TRIG
   #R_TRIG_SN(CLK := #Sn);   // R_TRIG
END_REGION
END_FUNCTION_BLOCK

FUNCTION_BLOCK "Elevator"   // FB6, LAD
{ S7_Optimized_Access := 'TRUE' }
VERSION : 0.1
   VAR_INPUT
      piano_richiesto : Int;
      exit_limit : Bool;
      enter_limit : Bool;
      position : Real;
      Sospendi : Bool;
      Forza : Bool;
   END_VAR
   VAR_OUTPUT
      pronto_ricevere : Bool;
      setpoint : Real;
      roll : Bool;
      motor1 : Bool;
      motor2 : Bool;
      motor3 : Bool;
   END_VAR
   VAR
      INIZ : Bool;
      p1 : Bool;
      p2 : Bool;
      p3 : Bool;
      p4 : Bool;
      p5 : Bool;
      p6 : Bool;
      p7 : Bool;
      t1 : Bool;
      t2 : Bool;
      t3 : Bool;
      t4 : Bool;
      t5 : Bool;
      t6 : Bool;
      t7 : Bool;
      R_TRIG_XL : R_TRIG;
      F_TRIG_XL : F_TRIG;
      F_TRIG_EL : F_TRIG;
      timer_p3 : TON_TIME;
      timer_p6 : TON_TIME;
      piano_mem : Int;
      quota_mem : Real;
      sub_out : Real;
      abs_out : Real;
   END_VAR
   VAR_TEMP   // added for the SCL form of the ladder/FBD networks
      _w1 : Bool;
   END_VAR
BEGIN

REGION Network 1: Inizializzazione
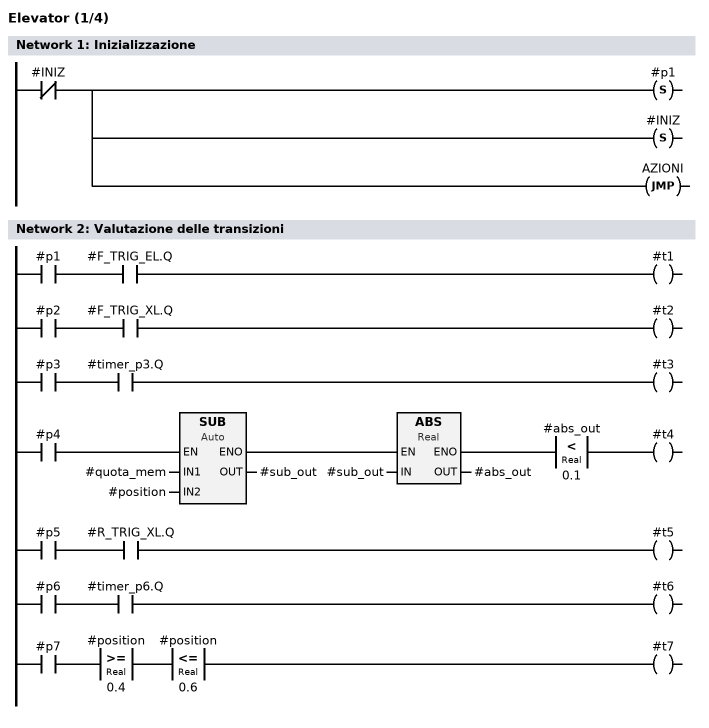
   RUNG wire#powerrail
      I_Contact( #INIZ )
      wire#w1
      S_Coil( #p1 )
   END_RUNG
   RUNG wire#w1
      S_Coil( #INIZ )
   END_RUNG
   RUNG wire#w1
      JumpCoil( AZIONI )
   END_RUNG
   // the same network as SCL:
   IF NOT #INIZ THEN #p1 := TRUE; END_IF;
   #_w1 := NOT #INIZ;
   IF #_w1 THEN
       #INIZ := TRUE;
       GOTO AZIONI;
   END_IF;
END_REGION

REGION Network 2: Valutazione delle transizioni
   RUNG wire#powerrail
      Contact( #p1 )
      Contact( #F_TRIG_EL.Q )
      Coil( #t1 )
   END_RUNG
   RUNG wire#powerrail
      Contact( #p2 )
      Contact( #F_TRIG_XL.Q )
      Coil( #t2 )
   END_RUNG
   RUNG wire#powerrail
      Contact( #p3 )
      Contact( #timer_p3.Q )
      Coil( #t3 )
   END_RUNG
   RUNG wire#powerrail
      Contact( #p4 )
      Sub(in1 := #quota_mem, in2 := #position, out => #sub_out)
      { S7_Templates := "SrcType := Real" } Abs(in := #sub_out, out => #abs_out)
      { S7_Templates := "SrcType := Real" } LT_Contact(in1 := #abs_out, in2 := 0.1)
      Coil( #t4 )
   END_RUNG
   RUNG wire#powerrail
      Contact( #p5 )
      Contact( #R_TRIG_XL.Q )
      Coil( #t5 )
   END_RUNG
   RUNG wire#powerrail
      Contact( #p6 )
      Contact( #timer_p6.Q )
      Coil( #t6 )
   END_RUNG
   RUNG wire#powerrail
      Contact( #p7 )
      { S7_Templates := "SrcType := Real" } GE_Contact(in1 := #position, in2 := 0.4)
      { S7_Templates := "SrcType := Real" } LE_Contact(in1 := #position, in2 := 0.6)
      Coil( #t7 )
   END_RUNG
   // the same network as SCL:
   #t1 := #p1 AND #F_TRIG_EL.Q;
   #t2 := #p2 AND #F_TRIG_XL.Q;
   #t3 := #p3 AND #timer_p3.Q;
   IF #p4 THEN
       #sub_out := #quota_mem - #position;
       #abs_out := ABS(#sub_out);
   END_IF;
   #t4 := #p4 AND (#abs_out < 0.1);
   #t5 := #p5 AND #R_TRIG_XL.Q;
   #t6 := #p6 AND #timer_p6.Q;
   #t7 := #p7 AND (#position >= 0.4) AND (#position <= 0.6);
END_REGION

REGION Network 3: Aggiornamento delle condizioni
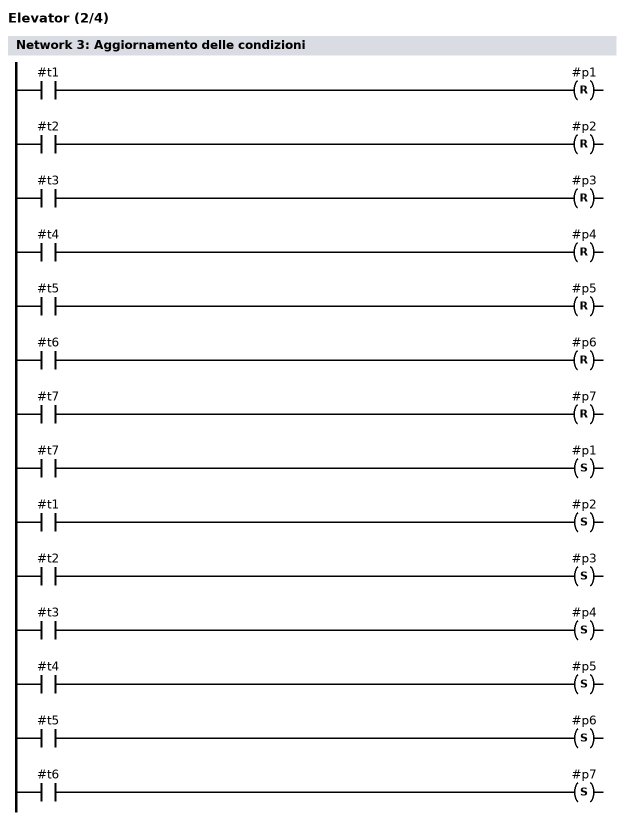
   RUNG wire#powerrail
      Contact( #t1 )
      R_Coil( #p1 )
   END_RUNG
   RUNG wire#powerrail
      Contact( #t2 )
      R_Coil( #p2 )
   END_RUNG
   RUNG wire#powerrail
      Contact( #t3 )
      R_Coil( #p3 )
   END_RUNG
   RUNG wire#powerrail
      Contact( #t4 )
      R_Coil( #p4 )
   END_RUNG
   RUNG wire#powerrail
      Contact( #t5 )
      R_Coil( #p5 )
   END_RUNG
   RUNG wire#powerrail
      Contact( #t6 )
      R_Coil( #p6 )
   END_RUNG
   RUNG wire#powerrail
      Contact( #t7 )
      R_Coil( #p7 )
   END_RUNG
   RUNG wire#powerrail
      Contact( #t7 )
      S_Coil( #p1 )
   END_RUNG
   RUNG wire#powerrail
      Contact( #t1 )
      S_Coil( #p2 )
   END_RUNG
   RUNG wire#powerrail
      Contact( #t2 )
      S_Coil( #p3 )
   END_RUNG
   RUNG wire#powerrail
      Contact( #t3 )
      S_Coil( #p4 )
   END_RUNG
   RUNG wire#powerrail
      Contact( #t4 )
      S_Coil( #p5 )
   END_RUNG
   RUNG wire#powerrail
      Contact( #t5 )
      S_Coil( #p6 )
   END_RUNG
   RUNG wire#powerrail
      Contact( #t6 )
      S_Coil( #p7 )
   END_RUNG
   // the same network as SCL:
   IF #t1 THEN #p1 := FALSE; END_IF;
   IF #t2 THEN #p2 := FALSE; END_IF;
   IF #t3 THEN #p3 := FALSE; END_IF;
   IF #t4 THEN #p4 := FALSE; END_IF;
   IF #t5 THEN #p5 := FALSE; END_IF;
   IF #t6 THEN #p6 := FALSE; END_IF;
   IF #t7 THEN
       #p7 := FALSE;
       #p1 := TRUE;
   END_IF;
   IF #t1 THEN #p2 := TRUE; END_IF;
   IF #t2 THEN #p3 := TRUE; END_IF;
   IF #t3 THEN #p4 := TRUE; END_IF;
   IF #t4 THEN #p5 := TRUE; END_IF;
   IF #t5 THEN #p6 := TRUE; END_IF;
   IF #t6 THEN #p7 := TRUE; END_IF;
END_REGION

REGION Network 4: Macroazioni di sospensione e forzatura alla fase 1 e sezione di esecuzione delle azioni
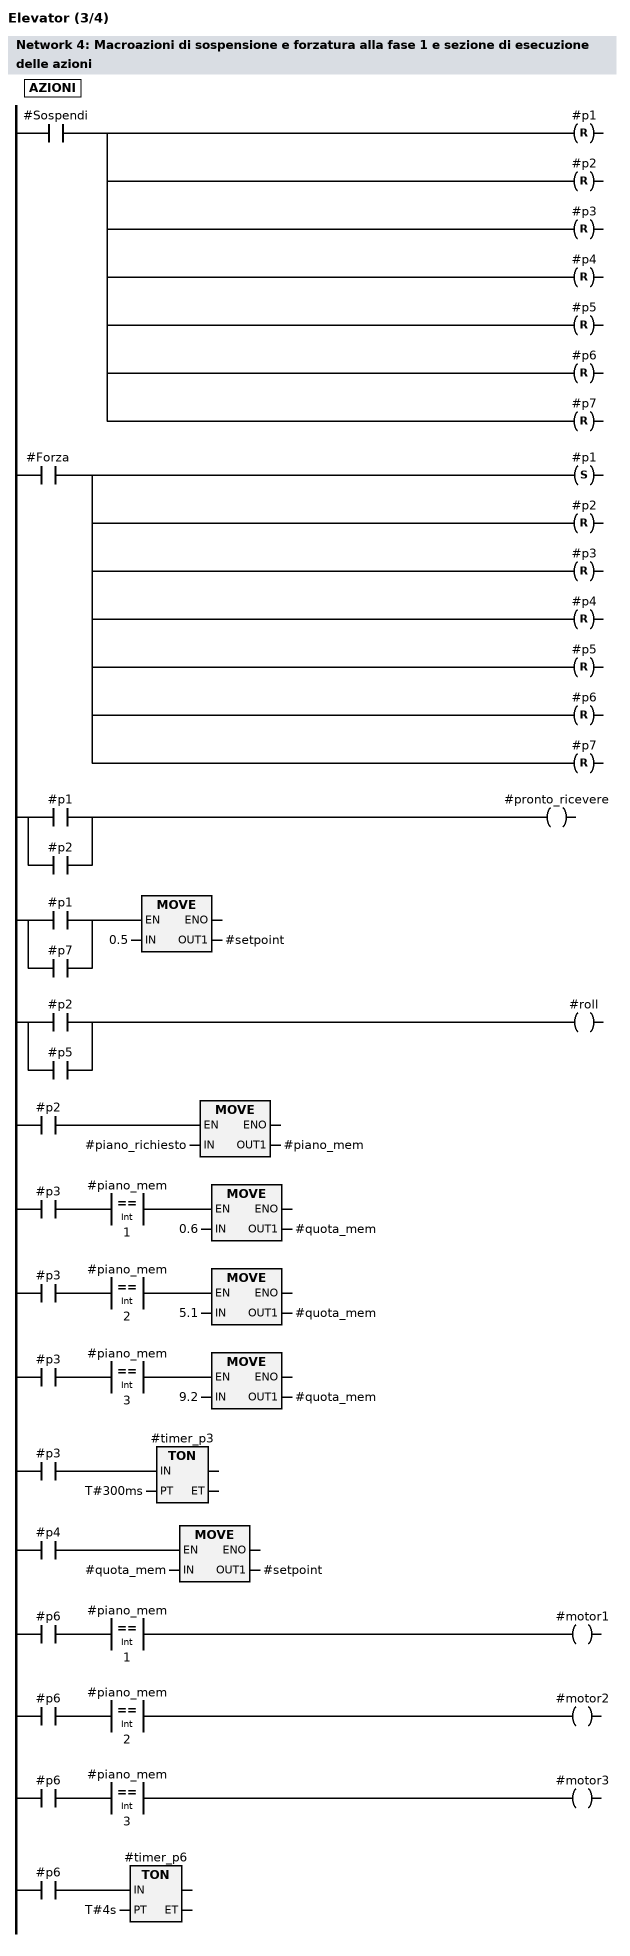
   AZIONI:
   IF #Sospendi THEN
       #p1 := FALSE;
       #p2 := FALSE;
       #p3 := FALSE;
       #p4 := FALSE;
       #p5 := FALSE;
       #p6 := FALSE;
       #p7 := FALSE;
   END_IF;
   IF #Forza THEN
       #p1 := TRUE;
       #p2 := FALSE;
       #p3 := FALSE;
       #p4 := FALSE;
       #p5 := FALSE;
       #p6 := FALSE;
       #p7 := FALSE;
   END_IF;
   #pronto_ricevere := #p1 OR #p2;
   IF #p1 OR #p7 THEN #setpoint := 0.5; END_IF;
   #roll := #p2 OR #p5;
   IF #p2 THEN #piano_mem := #piano_richiesto; END_IF;
   IF #p3 AND (#piano_mem = 1) THEN #quota_mem := 0.6; END_IF;
   IF #p3 AND (#piano_mem = 2) THEN #quota_mem := 5.1; END_IF;
   IF #p3 AND (#piano_mem = 3) THEN #quota_mem := 9.2; END_IF;
   #timer_p3(IN := #p3, PT := T#300ms);   // TON
   IF #p4 THEN #setpoint := #quota_mem; END_IF;
   #motor1 := #p6 AND (#piano_mem = 1);
   #motor2 := #p6 AND (#piano_mem = 2);
   #motor3 := #p6 AND (#piano_mem = 3);
   #timer_p6(IN := #p6, PT := T#4s);   // TON
END_REGION

REGION Network 5: Trigger
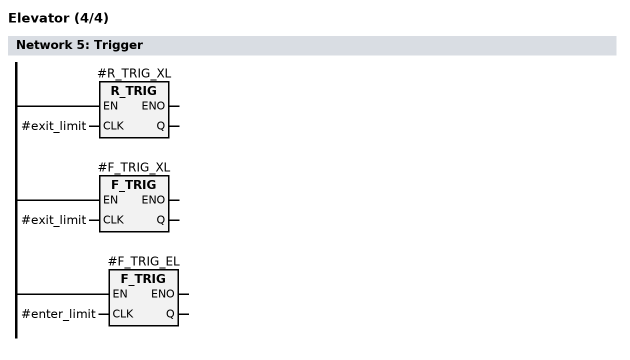
   #R_TRIG_XL(CLK := #exit_limit);   // R_TRIG
   #F_TRIG_XL(CLK := #exit_limit);   // F_TRIG
   #F_TRIG_EL(CLK := #enter_limit);   // F_TRIG
END_REGION
END_FUNCTION_BLOCK

FUNCTION_BLOCK "Pick-place"   // FB7, LAD
{ S7_Optimized_Access := 'TRUE' }
VERSION : 0.1
   VAR_INPUT
      X_position : Real;
      Y_position : Real;
      Z_position : Real;
      detected : Bool;
      work : Bool;
      Sospendi : Bool;
      Forza : Bool;
   END_VAR
   VAR_OUTPUT
      X_setpoint : Real;
      Y_setpoint : Real;
      Z_setpoint : Real;
      grab : Bool;
      work_finished : Bool;
   END_VAR
   VAR
      p1 : Bool;
      p2 : Bool;
      p3 : Bool;
      p4 : Bool;
      p5 : Bool;
      p6 : Bool;
      p7 : Bool;
      p8 : Bool;
      p9 : Bool;
      p10 : Bool;
      t1 : Bool;
      t2 : Bool;
      t3 : Bool;
      t4 : Bool;
      t5 : Bool;
      t6 : Bool;
      t7 : Bool;
      t8 : Bool;
      t9 : Bool;
      t10 : Bool;
      INIZ : Bool;
      timer_p3 : TON_TIME;
      timer_p4 : TON_TIME;
      timer_p8 : TON_TIME;
      sub_x : Real;
      sub_y : Real;
      sub_z : Real;
      abs_x : Real;
      abs_y : Real;
      abs_z : Real;
   END_VAR
   VAR_TEMP   // added for the SCL form of the ladder/FBD networks
      _w1 : Bool;
   END_VAR
BEGIN

REGION Network 1: Inizializzazione
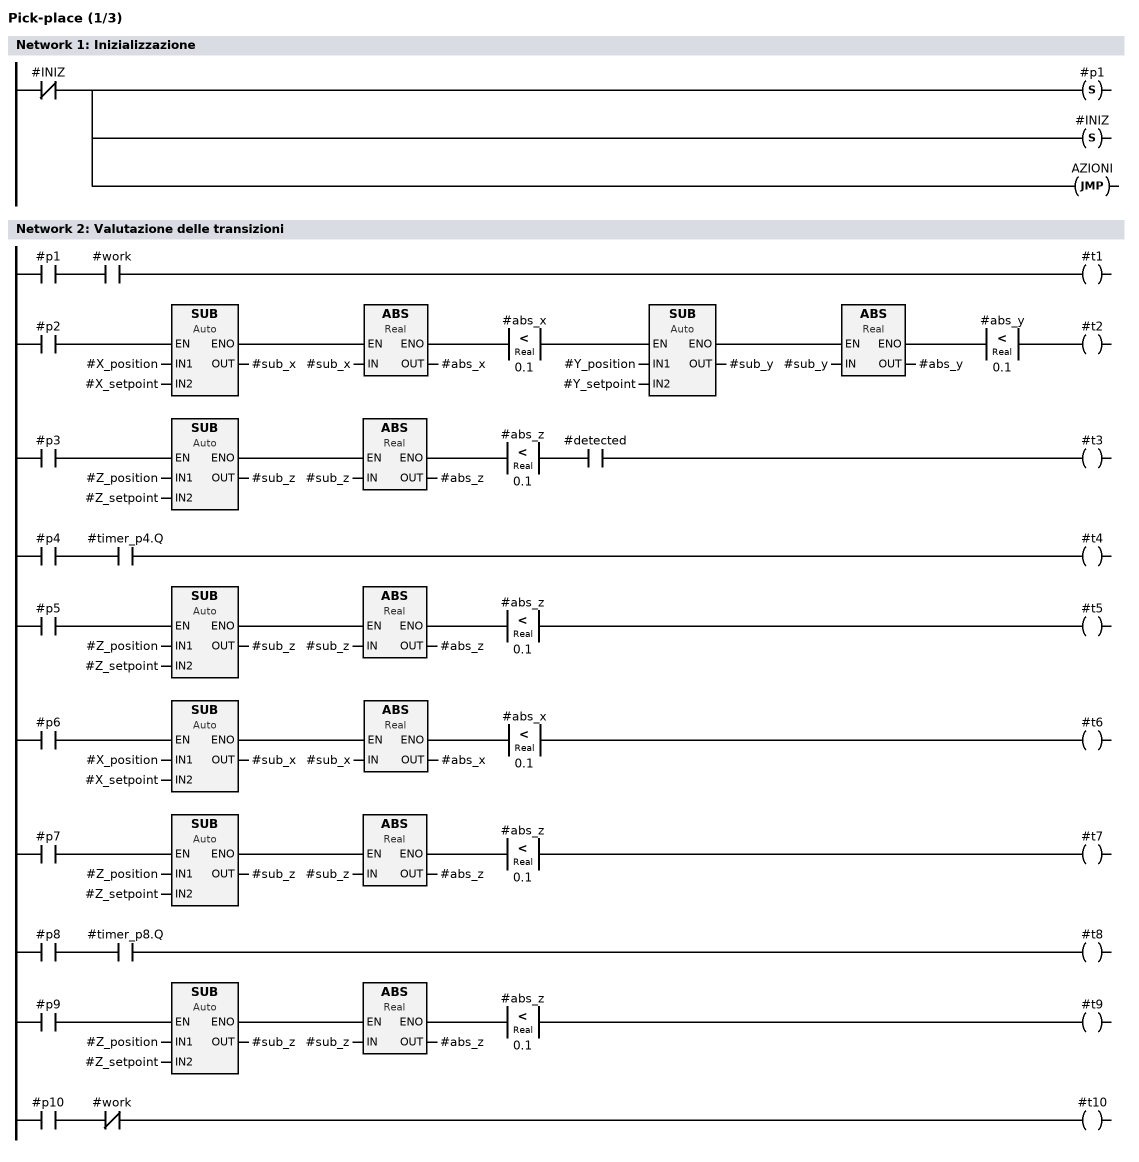
   RUNG wire#powerrail
      I_Contact( #INIZ )
      wire#w1
      S_Coil( #p1 )
   END_RUNG
   RUNG wire#w1
      S_Coil( #INIZ )
   END_RUNG
   RUNG wire#w1
      JumpCoil( AZIONI )
   END_RUNG
   // the same network as SCL:
   IF NOT #INIZ THEN #p1 := TRUE; END_IF;
   #_w1 := NOT #INIZ;
   IF #_w1 THEN
       #INIZ := TRUE;
       GOTO AZIONI;
   END_IF;
END_REGION

REGION Network 2: Valutazione delle transizioni
   RUNG wire#powerrail
      Contact( #p1 )
      Contact( #work )
      Coil( #t1 )
   END_RUNG
   RUNG wire#powerrail
      Contact( #p2 )
      Sub(in1 := #X_position, in2 := #X_setpoint, out => #sub_x)
      { S7_Templates := "SrcType := Real" } Abs(in := #sub_x, out => #abs_x)
      { S7_Templates := "SrcType := Real" } LT_Contact(in1 := #abs_x, in2 := 0.1)
      Sub(in1 := #Y_position, in2 := #Y_setpoint, out => #sub_y)
      { S7_Templates := "SrcType := Real" } Abs(in := #sub_y, out => #abs_y)
      { S7_Templates := "SrcType := Real" } LT_Contact(in1 := #abs_y, in2 := 0.1)
      Coil( #t2 )
   END_RUNG
   RUNG wire#powerrail
      Contact( #p3 )
      Sub(in1 := #Z_position, in2 := #Z_setpoint, out => #sub_z)
      { S7_Templates := "SrcType := Real" } Abs(in := #sub_z, out => #abs_z)
      { S7_Templates := "SrcType := Real" } LT_Contact(in1 := #abs_z, in2 := 0.1)
      Contact( #detected )
      Coil( #t3 )
   END_RUNG
   RUNG wire#powerrail
      Contact( #p4 )
      Contact( #timer_p4.Q )
      Coil( #t4 )
   END_RUNG
   RUNG wire#powerrail
      Contact( #p5 )
      Sub(in1 := #Z_position, in2 := #Z_setpoint, out => #sub_z)
      { S7_Templates := "SrcType := Real" } Abs(in := #sub_z, out => #abs_z)
      { S7_Templates := "SrcType := Real" } LT_Contact(in1 := #abs_z, in2 := 0.1)
      Coil( #t5 )
   END_RUNG
   RUNG wire#powerrail
      Contact( #p6 )
      Sub(in1 := #X_position, in2 := #X_setpoint, out => #sub_x)
      { S7_Templates := "SrcType := Real" } Abs(in := #sub_x, out => #abs_x)
      { S7_Templates := "SrcType := Real" } LT_Contact(in1 := #abs_x, in2 := 0.1)
      Coil( #t6 )
   END_RUNG
   RUNG wire#powerrail
      Contact( #p7 )
      Sub(in1 := #Z_position, in2 := #Z_setpoint, out => #sub_z)
      { S7_Templates := "SrcType := Real" } Abs(in := #sub_z, out => #abs_z)
      { S7_Templates := "SrcType := Real" } LT_Contact(in1 := #abs_z, in2 := 0.1)
      Coil( #t7 )
   END_RUNG
   RUNG wire#powerrail
      Contact( #p8 )
      Contact( #timer_p8.Q )
      Coil( #t8 )
   END_RUNG
   RUNG wire#powerrail
      Contact( #p9 )
      Sub(in1 := #Z_position, in2 := #Z_setpoint, out => #sub_z)
      { S7_Templates := "SrcType := Real" } Abs(in := #sub_z, out => #abs_z)
      { S7_Templates := "SrcType := Real" } LT_Contact(in1 := #abs_z, in2 := 0.1)
      Coil( #t9 )
   END_RUNG
   RUNG wire#powerrail
      Contact( #p10 )
      I_Contact( #work )
      Coil( #t10 )
   END_RUNG
   // the same network as SCL:
   #t1 := #p1 AND #work;
   IF #p2 THEN
       #sub_x := #X_position - #X_setpoint;
       #abs_x := ABS(#sub_x);
   END_IF;
   #_w1 := #p2 AND (#abs_x < 0.1);
   IF #_w1 THEN
       #sub_y := #Y_position - #Y_setpoint;
       #abs_y := ABS(#sub_y);
   END_IF;
   #t2 := #_w1 AND (#abs_y < 0.1);
   IF #p3 THEN
       #sub_z := #Z_position - #Z_setpoint;
       #abs_z := ABS(#sub_z);
   END_IF;
   #t3 := #p3 AND (#abs_z < 0.1) AND #detected;
   #t4 := #p4 AND #timer_p4.Q;
   IF #p5 THEN
       #sub_z := #Z_position - #Z_setpoint;
       #abs_z := ABS(#sub_z);
   END_IF;
   #t5 := #p5 AND (#abs_z < 0.1);
   IF #p6 THEN
       #sub_x := #X_position - #X_setpoint;
       #abs_x := ABS(#sub_x);
   END_IF;
   #t6 := #p6 AND (#abs_x < 0.1);
   IF #p7 THEN
       #sub_z := #Z_position - #Z_setpoint;
       #abs_z := ABS(#sub_z);
   END_IF;
   #t7 := #p7 AND (#abs_z < 0.1);
   #t8 := #p8 AND #timer_p8.Q;
   IF #p9 THEN
       #sub_z := #Z_position - #Z_setpoint;
       #abs_z := ABS(#sub_z);
   END_IF;
   #t9 := #p9 AND (#abs_z < 0.1);
   #t10 := #p10 AND NOT #work;
END_REGION

REGION Network 3: Aggiornamento delle condizioni
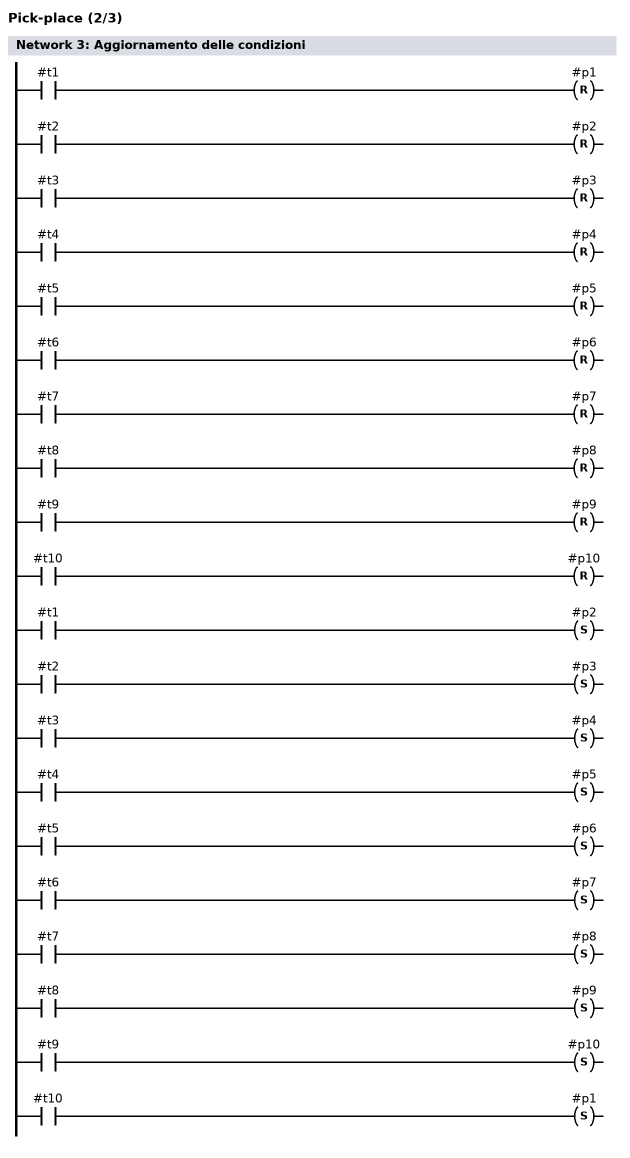
   RUNG wire#powerrail
      Contact( #t1 )
      R_Coil( #p1 )
   END_RUNG
   RUNG wire#powerrail
      Contact( #t2 )
      R_Coil( #p2 )
   END_RUNG
   RUNG wire#powerrail
      Contact( #t3 )
      R_Coil( #p3 )
   END_RUNG
   RUNG wire#powerrail
      Contact( #t4 )
      R_Coil( #p4 )
   END_RUNG
   RUNG wire#powerrail
      Contact( #t5 )
      R_Coil( #p5 )
   END_RUNG
   RUNG wire#powerrail
      Contact( #t6 )
      R_Coil( #p6 )
   END_RUNG
   RUNG wire#powerrail
      Contact( #t7 )
      R_Coil( #p7 )
   END_RUNG
   RUNG wire#powerrail
      Contact( #t8 )
      R_Coil( #p8 )
   END_RUNG
   RUNG wire#powerrail
      Contact( #t9 )
      R_Coil( #p9 )
   END_RUNG
   RUNG wire#powerrail
      Contact( #t10 )
      R_Coil( #p10 )
   END_RUNG
   RUNG wire#powerrail
      Contact( #t1 )
      S_Coil( #p2 )
   END_RUNG
   RUNG wire#powerrail
      Contact( #t2 )
      S_Coil( #p3 )
   END_RUNG
   RUNG wire#powerrail
      Contact( #t3 )
      S_Coil( #p4 )
   END_RUNG
   RUNG wire#powerrail
      Contact( #t4 )
      S_Coil( #p5 )
   END_RUNG
   RUNG wire#powerrail
      Contact( #t5 )
      S_Coil( #p6 )
   END_RUNG
   RUNG wire#powerrail
      Contact( #t6 )
      S_Coil( #p7 )
   END_RUNG
   RUNG wire#powerrail
      Contact( #t7 )
      S_Coil( #p8 )
   END_RUNG
   RUNG wire#powerrail
      Contact( #t8 )
      S_Coil( #p9 )
   END_RUNG
   RUNG wire#powerrail
      Contact( #t9 )
      S_Coil( #p10 )
   END_RUNG
   RUNG wire#powerrail
      Contact( #t10 )
      S_Coil( #p1 )
   END_RUNG
   // the same network as SCL:
   IF #t1 THEN #p1 := FALSE; END_IF;
   IF #t2 THEN #p2 := FALSE; END_IF;
   IF #t3 THEN #p3 := FALSE; END_IF;
   IF #t4 THEN #p4 := FALSE; END_IF;
   IF #t5 THEN #p5 := FALSE; END_IF;
   IF #t6 THEN #p6 := FALSE; END_IF;
   IF #t7 THEN #p7 := FALSE; END_IF;
   IF #t8 THEN #p8 := FALSE; END_IF;
   IF #t9 THEN #p9 := FALSE; END_IF;
   IF #t10 THEN #p10 := FALSE; END_IF;
   IF #t1 THEN #p2 := TRUE; END_IF;
   IF #t2 THEN #p3 := TRUE; END_IF;
   IF #t3 THEN #p4 := TRUE; END_IF;
   IF #t4 THEN #p5 := TRUE; END_IF;
   IF #t5 THEN #p6 := TRUE; END_IF;
   IF #t6 THEN #p7 := TRUE; END_IF;
   IF #t7 THEN #p8 := TRUE; END_IF;
   IF #t8 THEN #p9 := TRUE; END_IF;
   IF #t9 THEN #p10 := TRUE; END_IF;
   IF #t10 THEN #p1 := TRUE; END_IF;
END_REGION

REGION Network 4: Macroazioni di sospensione e forzatura alla fase 1 e sezione di esecuzione delle azioni
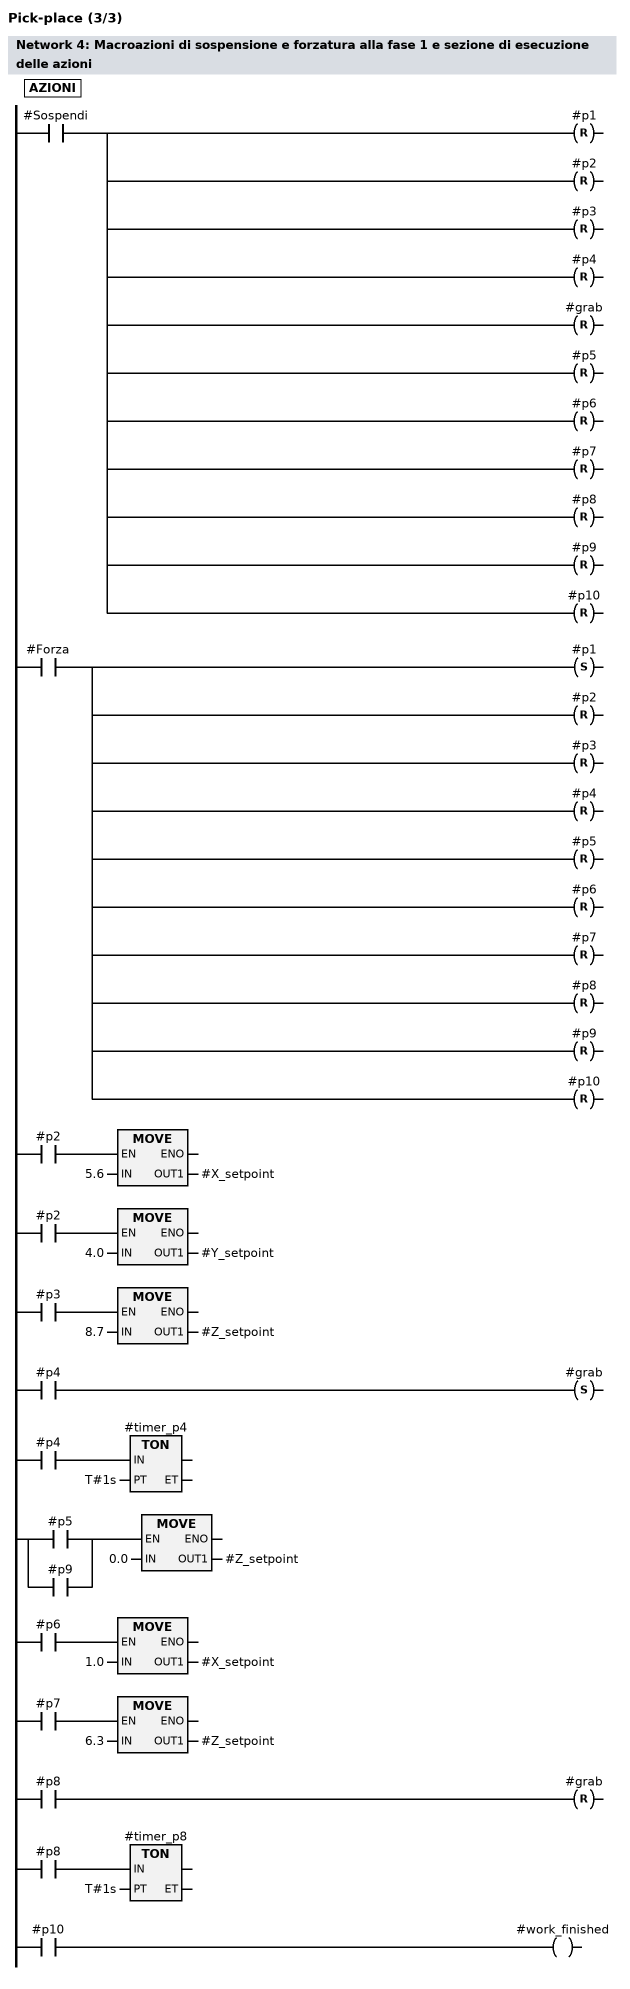
   AZIONI:
   IF #Sospendi THEN
       #p1 := FALSE;
       #p2 := FALSE;
       #p3 := FALSE;
       #p4 := FALSE;
       #grab := FALSE;
       #p5 := FALSE;
       #p6 := FALSE;
       #p7 := FALSE;
       #p8 := FALSE;
       #p9 := FALSE;
       #p10 := FALSE;
   END_IF;
   IF #Forza THEN
       #p1 := TRUE;
       #p2 := FALSE;
       #p3 := FALSE;
       #p4 := FALSE;
       #p5 := FALSE;
       #p6 := FALSE;
       #p7 := FALSE;
       #p8 := FALSE;
       #p9 := FALSE;
       #p10 := FALSE;
   END_IF;
   IF #p2 THEN
       #X_setpoint := 5.6;
       #Y_setpoint := 4.0;
   END_IF;
   IF #p3 THEN #Z_setpoint := 8.7; END_IF;
   IF #p4 THEN #grab := TRUE; END_IF;
   #timer_p4(IN := #p4, PT := T#1s);   // TON
   IF #p5 OR #p9 THEN #Z_setpoint := 0.0; END_IF;
   IF #p6 THEN #X_setpoint := 1.0; END_IF;
   IF #p7 THEN #Z_setpoint := 6.3; END_IF;
   IF #p8 THEN #grab := FALSE; END_IF;
   #timer_p8(IN := #p8, PT := T#1s);   // TON
   #work_finished := #p10;
END_REGION
END_FUNCTION_BLOCK

FUNCTION "MHJ-PLC-Lab-Function-S71200" : Void   // FC9000, SCL
{ S7_Optimized_Access := 'TRUE' }
VERSION : 0.1
   VAR_TEMP
      rdTimeReturn : Int;
      outputTime : DTL;
      SyncVal : Byte;
      forVal : Int;
      forVal_2 : Int;
      Value : Byte;
   END_VAR
   VAR CONSTANT
      CompVal : Byte := 16#34;
      Value_01 : Byte := 16#11;
      Value_01_DW : DWord := 16#A165_D992;
      Value_02_DW : DWord := 16#58BE_4401;
   END_VAR
BEGIN

   #Value:=PEEK(area := 16#82,
        dbNumber := 0,
        byteOffset := 511);
   #Value := #Value + 1;

   POKE(area := 16#82,
        dbNumber := 0,
        byteOffset := 511,
        value := #Value);

   POKE(area:=16#81,
        dbNumber:=0,
        byteOffset:=1016,
        value:=#Value_01_DW);
   POKE(area := 16#81,
        dbNumber := 0,
        byteOffset := 1020,
        value := #Value_02_DW);

   POKE(area := 16#81,
        dbNumber := 0,
        byteOffset := 511,
        value := B#16#00);

   FOR #forVal := 0 TO 120 DO
       FOR #forVal_2:=0 TO 10 DO
           #rdTimeReturn:=RD_SYS_T(#outputTime);
           #rdTimeReturn := WR_SYS_T(#outputTime);
           #rdTimeReturn := RD_SYS_T(#outputTime);
           #rdTimeReturn := WR_SYS_T(#outputTime);
       END_FOR;
       #SyncVal:= PEEK(area := 16#81,
                      dbNumber := 0,
                      byteOffset := 511);
       IF #SyncVal = #CompVal THEN
          GOTO M_1;
       END_IF;
   END_FOR;
   RETURN;

   M_1:
   POKE(area := 16#81,
        dbNumber := 0,
        byteOffset := 511,
        value := B#16#0);
END_FUNCTION

ORGANIZATION_BLOCK "Main"   // OB1, LAD, ProgramCycle
TITLE = "Main Program Sweep (Cycle)"
{ S7_Optimized_Access := 'TRUE' }
VERSION : 0.1
   VAR_INPUT
      Initial_Call : Bool;   // Initial call of this OB
      Remanence : Bool;   // =True, if remanent data are available
   END_VAR
BEGIN

REGION Network 1
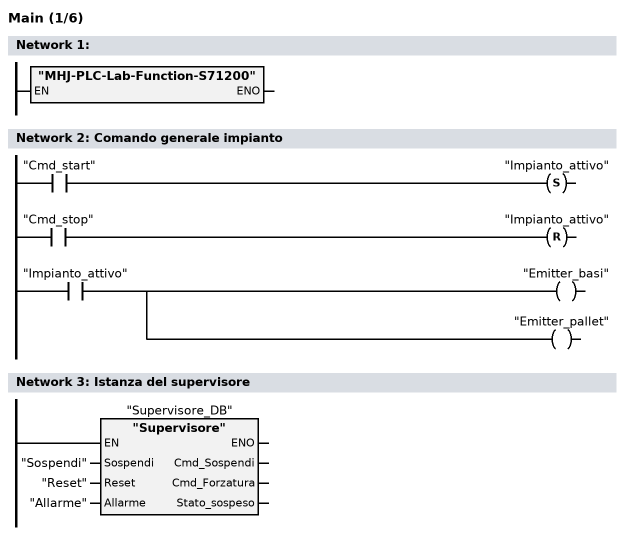
   RUNG wire#powerrail
      "MHJ-PLC-Lab-Function-S71200"()
   END_RUNG
   // the same network as SCL:
   "MHJ-PLC-Lab-Function-S71200"();
END_REGION

REGION Network 2: Comando generale impianto
   RUNG wire#powerrail
      Contact( "Cmd_start" )
      S_Coil( "Impianto_attivo" )
   END_RUNG
   RUNG wire#powerrail
      Contact( "Cmd_stop" )
      R_Coil( "Impianto_attivo" )
   END_RUNG
   RUNG wire#powerrail
      Contact( "Impianto_attivo" )
      wire#w1
      Coil( "Emitter_basi" )
   END_RUNG
   RUNG wire#w1
      Coil( "Emitter_pallet" )
   END_RUNG
   // the same network as SCL:
   IF "Cmd_start" THEN "Impianto_attivo" := TRUE; END_IF;
   IF "Cmd_stop" THEN "Impianto_attivo" := FALSE; END_IF;
   "Emitter_basi" := "Impianto_attivo";
   "Emitter_pallet" := "Impianto_attivo";
END_REGION

REGION Network 3: Istanza del supervisore
   RUNG wire#powerrail
      "Supervisore_DB"(Sospendi := "Sospendi", Reset := "Reset", Allarme := "Allarme", Cmd_Sospendi =>, Cmd_Forzatura =>, Stato_sospeso =>)
   END_RUNG
   // the same network as SCL:
   "Supervisore_DB"(Sospendi := "Sospendi", Reset := "Reset", Allarme := "Allarme");   // "Supervisore"
END_REGION

REGION Network 4: Impianto generale
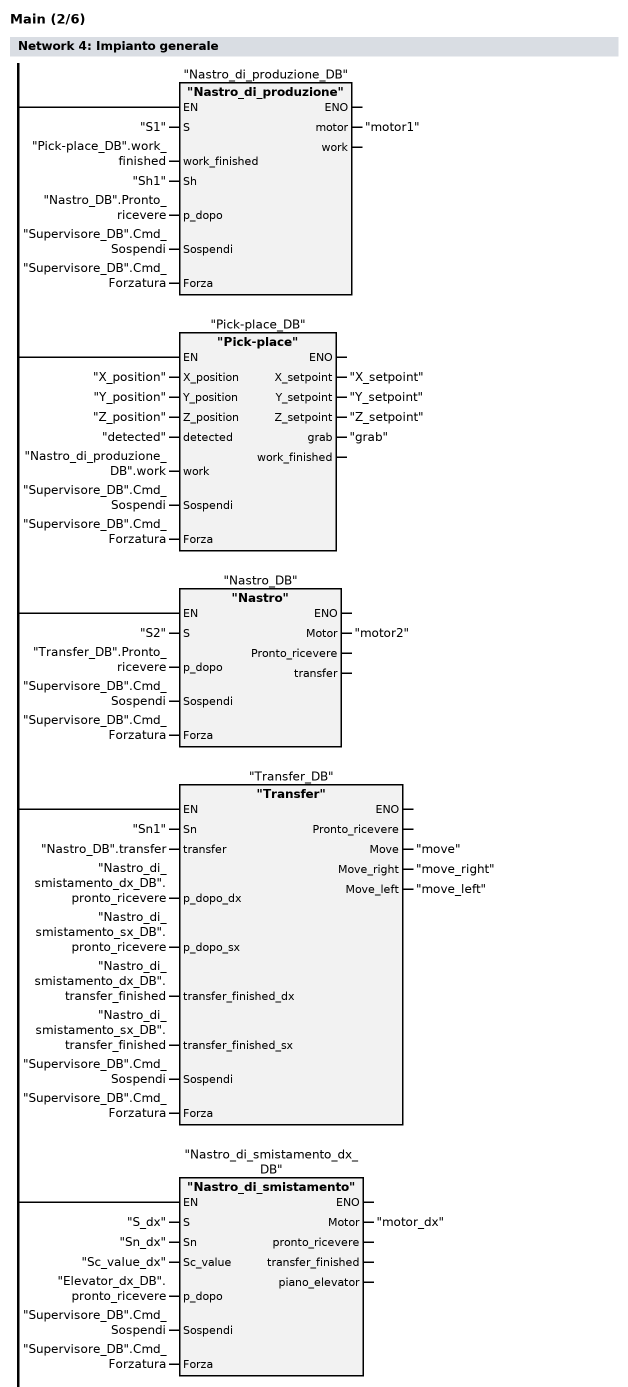
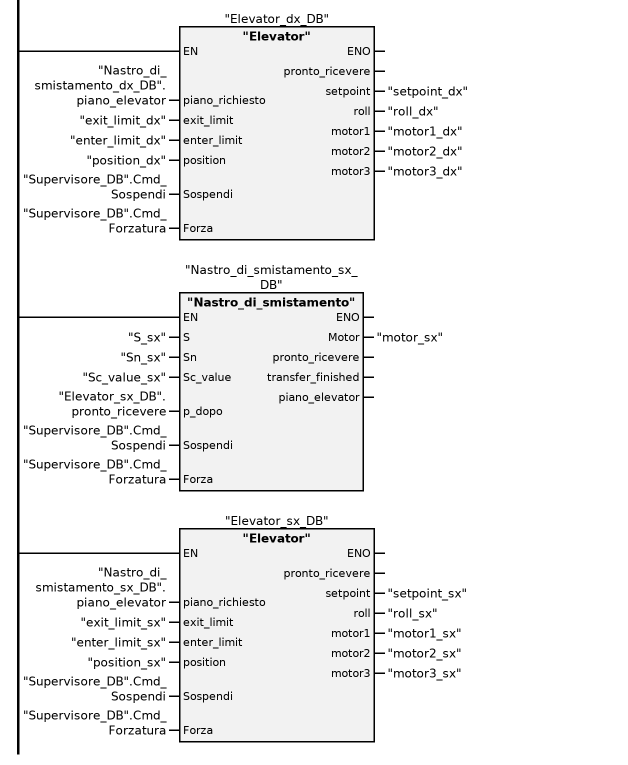
   RUNG wire#powerrail
      "Nastro_di_produzione_DB"(S := "S1", work_finished := "Pick-place_DB".work_finished, Sh := "Sh1", p_dopo := "Nastro_DB".Pronto_ricevere, Sospendi := "Supervisore_DB".Cmd_Sospendi, Forza := "Supervisore_DB".Cmd_Forzatura, motor => "motor1", work =>)
   END_RUNG
   RUNG wire#powerrail
      "Pick-place_DB"(X_position := "X_position", Y_position := "Y_position", Z_position := "Z_position", detected := "detected", work := "Nastro_di_produzione_DB".work, Sospendi := "Supervisore_DB".Cmd_Sospendi, Forza := "Supervisore_DB".Cmd_Forzatura, X_setpoint => "X_setpoint", Y_setpoint => "Y_setpoint", Z_setpoint => "Z_setpoint", grab => "grab", work_finished =>)
   END_RUNG
   RUNG wire#powerrail
      "Nastro_DB"(S := "S2", p_dopo := "Transfer_DB".Pronto_ricevere, Sospendi := "Supervisore_DB".Cmd_Sospendi, Forza := "Supervisore_DB".Cmd_Forzatura, Motor => "motor2", Pronto_ricevere =>, transfer =>)
   END_RUNG
   RUNG wire#powerrail
      "Transfer_DB"(Sn := "Sn1", transfer := "Nastro_DB".transfer, p_dopo_dx := "Nastro_di_smistamento_dx_DB".pronto_ricevere, p_dopo_sx := "Nastro_di_smistamento_sx_DB".pronto_ricevere, transfer_finished_dx := "Nastro_di_smistamento_dx_DB".transfer_finished, transfer_finished_sx := "Nastro_di_smistamento_sx_DB".transfer_finished, Sospendi := "Supervisore_DB".Cmd_Sospendi, Forza := "Supervisore_DB".Cmd_Forzatura, Pronto_ricevere =>, Move => "move", Move_right => "move_right", Move_left => "move_left")
   END_RUNG
   RUNG wire#powerrail
      "Nastro_di_smistamento_dx_DB"(S := "S_dx", Sn := "Sn_dx", Sc_value := "Sc_value_dx", p_dopo := "Elevator_dx_DB".pronto_ricevere, Sospendi := "Supervisore_DB".Cmd_Sospendi, Forza := "Supervisore_DB".Cmd_Forzatura, Motor => "motor_dx", pronto_ricevere =>, transfer_finished =>, piano_elevator =>)
   END_RUNG
   RUNG wire#powerrail
      "Elevator_dx_DB"(piano_richiesto := "Nastro_di_smistamento_dx_DB".piano_elevator, exit_limit := "exit_limit_dx", enter_limit := "enter_limit_dx", position := "position_dx", Sospendi := "Supervisore_DB".Cmd_Sospendi, Forza := "Supervisore_DB".Cmd_Forzatura, pronto_ricevere =>, setpoint => "setpoint_dx", roll => "roll_dx", motor1 => "motor1_dx", motor2 => "motor2_dx", motor3 => "motor3_dx")
   END_RUNG
   RUNG wire#powerrail
      "Nastro_di_smistamento_sx_DB"(S := "S_sx", Sn := "Sn_sx", Sc_value := "Sc_value_sx", p_dopo := "Elevator_sx_DB".pronto_ricevere, Sospendi := "Supervisore_DB".Cmd_Sospendi, Forza := "Supervisore_DB".Cmd_Forzatura, Motor => "motor_sx", pronto_ricevere =>, transfer_finished =>, piano_elevator =>)
   END_RUNG
   RUNG wire#powerrail
      "Elevator_sx_DB"(piano_richiesto := "Nastro_di_smistamento_sx_DB".piano_elevator, exit_limit := "exit_limit_sx", enter_limit := "enter_limit_sx", position := "position_sx", Sospendi := "Supervisore_DB".Cmd_Sospendi, Forza := "Supervisore_DB".Cmd_Forzatura, pronto_ricevere =>, setpoint => "setpoint_sx", roll => "roll_sx", motor1 => "motor1_sx", motor2 => "motor2_sx", motor3 => "motor3_sx")
   END_RUNG
   // the same network as SCL:
   "Nastro_di_produzione_DB"(S := "S1",   // "Nastro_di_produzione"
                           work_finished := "Pick-place_DB".work_finished,
                           Sh := "Sh1",
                           p_dopo := "Nastro_DB".Pronto_ricevere,
                           Sospendi := "Supervisore_DB".Cmd_Sospendi,
                           Forza := "Supervisore_DB".Cmd_Forzatura,
                           motor => "motor1");
   "Pick-place_DB"(X_position := "X_position",   // "Pick-place"
                   Y_position := "Y_position",
                   Z_position := "Z_position",
                   detected := "detected",
                   work := "Nastro_di_produzione_DB".work,
                   Sospendi := "Supervisore_DB".Cmd_Sospendi,
                   Forza := "Supervisore_DB".Cmd_Forzatura,
                   X_setpoint => "X_setpoint",
                   Y_setpoint => "Y_setpoint",
                   Z_setpoint => "Z_setpoint",
                   grab => "grab");
   "Nastro_DB"(S := "S2",   // "Nastro"
               p_dopo := "Transfer_DB".Pronto_ricevere,
               Sospendi := "Supervisore_DB".Cmd_Sospendi,
               Forza := "Supervisore_DB".Cmd_Forzatura,
               Motor => "motor2");
   "Transfer_DB"(Sn := "Sn1",   // "Transfer"
                 transfer := "Nastro_DB".transfer,
                 p_dopo_dx := "Nastro_di_smistamento_dx_DB".pronto_ricevere,
                 p_dopo_sx := "Nastro_di_smistamento_sx_DB".pronto_ricevere,
                 transfer_finished_dx := "Nastro_di_smistamento_dx_DB".transfer_finished,
                 transfer_finished_sx := "Nastro_di_smistamento_sx_DB".transfer_finished,
                 Sospendi := "Supervisore_DB".Cmd_Sospendi,
                 Forza := "Supervisore_DB".Cmd_Forzatura,
                 Move => "move",
                 Move_right => "move_right",
                 Move_left => "move_left");
   "Nastro_di_smistamento_dx_DB"(S := "S_dx",   // "Nastro_di_smistamento"
                           Sn := "Sn_dx",
                           Sc_value := "Sc_value_dx",
                           p_dopo := "Elevator_dx_DB".pronto_ricevere,
                           Sospendi := "Supervisore_DB".Cmd_Sospendi,
                           Forza := "Supervisore_DB".Cmd_Forzatura,
                           Motor => "motor_dx");
   "Elevator_dx_DB"(piano_richiesto := "Nastro_di_smistamento_dx_DB".piano_elevator,   // "Elevator"
                    exit_limit := "exit_limit_dx",
                    enter_limit := "enter_limit_dx",
                    position := "position_dx",
                    Sospendi := "Supervisore_DB".Cmd_Sospendi,
                    Forza := "Supervisore_DB".Cmd_Forzatura,
                    setpoint => "setpoint_dx",
                    roll => "roll_dx",
                    motor1 => "motor1_dx",
                    motor2 => "motor2_dx",
                    motor3 => "motor3_dx");
   "Nastro_di_smistamento_sx_DB"(S := "S_sx",   // "Nastro_di_smistamento"
                           Sn := "Sn_sx",
                           Sc_value := "Sc_value_sx",
                           p_dopo := "Elevator_sx_DB".pronto_ricevere,
                           Sospendi := "Supervisore_DB".Cmd_Sospendi,
                           Forza := "Supervisore_DB".Cmd_Forzatura,
                           Motor => "motor_sx");
   "Elevator_sx_DB"(piano_richiesto := "Nastro_di_smistamento_sx_DB".piano_elevator,   // "Elevator"
                    exit_limit := "exit_limit_sx",
                    enter_limit := "enter_limit_sx",
                    position := "position_sx",
                    Sospendi := "Supervisore_DB".Cmd_Sospendi,
                    Forza := "Supervisore_DB".Cmd_Forzatura,
                    setpoint => "setpoint_sx",
                    roll => "roll_sx",
                    motor1 => "motor1_sx",
                    motor2 => "motor2_sx",
                    motor3 => "motor3_sx");
END_REGION

REGION Network 5: Istanze di R_TRIG per conteggio e allarme
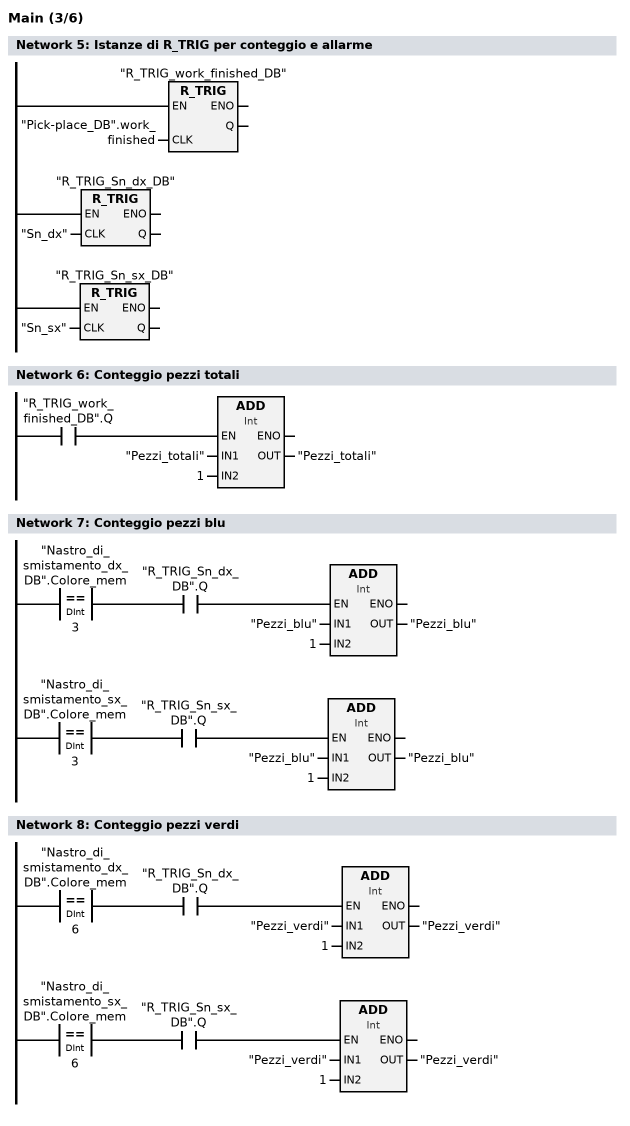
   "R_TRIG_work_finished_DB"(CLK := "Pick-place_DB".work_finished);   // R_TRIG
   "R_TRIG_Sn_dx_DB"(CLK := "Sn_dx");   // R_TRIG
   "R_TRIG_Sn_sx_DB"(CLK := "Sn_sx");   // R_TRIG
END_REGION

REGION Network 6: Conteggio pezzi totali
   RUNG wire#powerrail
      Contact( "R_TRIG_work_finished_DB".Q )
      { S7_Templates := "SrcType := Int" } Add(in1 := "Pezzi_totali", in2 := 1, out => "Pezzi_totali")
   END_RUNG
   // the same network as SCL:
   IF "R_TRIG_work_finished_DB".Q THEN "Pezzi_totali" := "Pezzi_totali" + 1; END_IF;
END_REGION

REGION Network 7: Conteggio pezzi blu
   RUNG wire#powerrail
      { S7_Templates := "SrcType := DInt" } EQ_Contact(in1 := "Nastro_di_smistamento_dx_DB".Colore_mem, in2 := 3)
      Contact( "R_TRIG_Sn_dx_DB".Q )
      { S7_Templates := "SrcType := Int" } Add(in1 := "Pezzi_blu", in2 := 1, out => "Pezzi_blu")
   END_RUNG
   RUNG wire#powerrail
      { S7_Templates := "SrcType := DInt" } EQ_Contact(in1 := "Nastro_di_smistamento_sx_DB".Colore_mem, in2 := 3)
      Contact( "R_TRIG_Sn_sx_DB".Q )
      { S7_Templates := "SrcType := Int" } Add(in1 := "Pezzi_blu", in2 := 1, out => "Pezzi_blu")
   END_RUNG
   // the same network as SCL:
   IF ("Nastro_di_smistamento_dx_DB".Colore_mem = 3) AND "R_TRIG_Sn_dx_DB".Q THEN
       "Pezzi_blu" := "Pezzi_blu" + 1;
   END_IF;
   IF ("Nastro_di_smistamento_sx_DB".Colore_mem = 3) AND "R_TRIG_Sn_sx_DB".Q THEN
       "Pezzi_blu" := "Pezzi_blu" + 1;
   END_IF;
END_REGION

REGION Network 8: Conteggio pezzi verdi
   RUNG wire#powerrail
      { S7_Templates := "SrcType := DInt" } EQ_Contact(in1 := "Nastro_di_smistamento_dx_DB".Colore_mem, in2 := 6)
      Contact( "R_TRIG_Sn_dx_DB".Q )
      { S7_Templates := "SrcType := Int" } Add(in1 := "Pezzi_verdi", in2 := 1, out => "Pezzi_verdi")
   END_RUNG
   RUNG wire#powerrail
      { S7_Templates := "SrcType := DInt" } EQ_Contact(in1 := "Nastro_di_smistamento_sx_DB".Colore_mem, in2 := 6)
      Contact( "R_TRIG_Sn_sx_DB".Q )
      { S7_Templates := "SrcType := Int" } Add(in1 := "Pezzi_verdi", in2 := 1, out => "Pezzi_verdi")
   END_RUNG
   // the same network as SCL:
   IF ("Nastro_di_smistamento_dx_DB".Colore_mem = 6) AND "R_TRIG_Sn_dx_DB".Q THEN
       "Pezzi_verdi" := "Pezzi_verdi" + 1;
   END_IF;
   IF ("Nastro_di_smistamento_sx_DB".Colore_mem = 6) AND "R_TRIG_Sn_sx_DB".Q THEN
       "Pezzi_verdi" := "Pezzi_verdi" + 1;
   END_IF;
END_REGION

REGION Network 9: Conteggio pezzi grigi
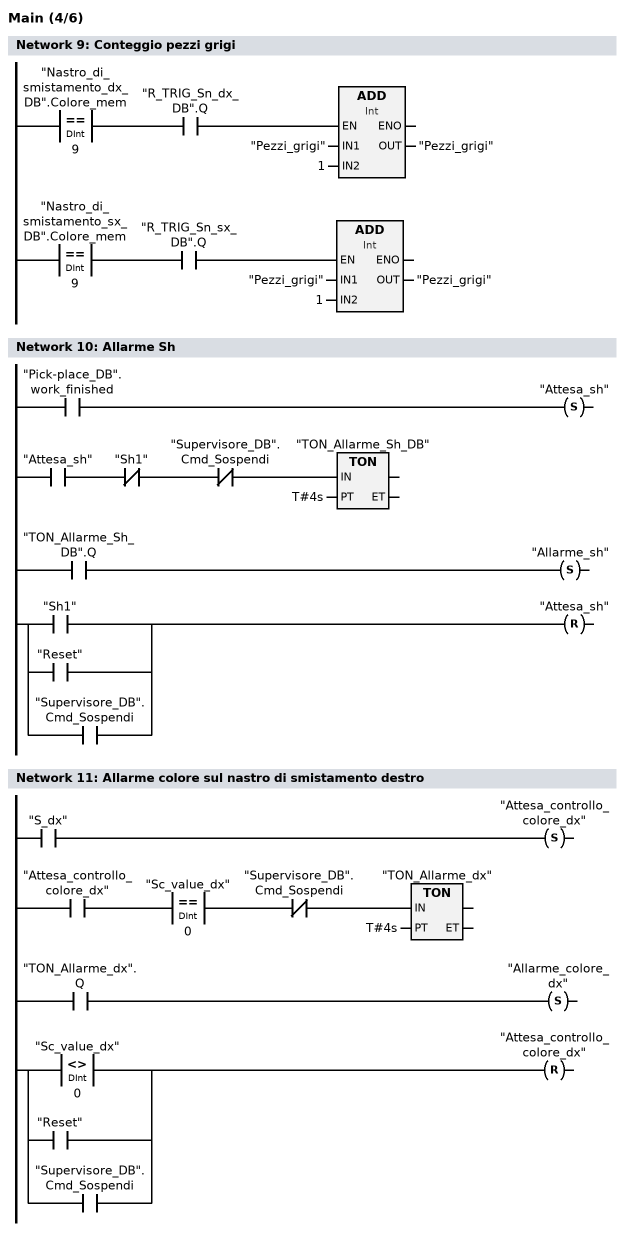
   RUNG wire#powerrail
      { S7_Templates := "SrcType := DInt" } EQ_Contact(in1 := "Nastro_di_smistamento_dx_DB".Colore_mem, in2 := 9)
      Contact( "R_TRIG_Sn_dx_DB".Q )
      { S7_Templates := "SrcType := Int" } Add(in1 := "Pezzi_grigi", in2 := 1, out => "Pezzi_grigi")
   END_RUNG
   RUNG wire#powerrail
      { S7_Templates := "SrcType := DInt" } EQ_Contact(in1 := "Nastro_di_smistamento_sx_DB".Colore_mem, in2 := 9)
      Contact( "R_TRIG_Sn_sx_DB".Q )
      { S7_Templates := "SrcType := Int" } Add(in1 := "Pezzi_grigi", in2 := 1, out => "Pezzi_grigi")
   END_RUNG
   // the same network as SCL:
   IF ("Nastro_di_smistamento_dx_DB".Colore_mem = 9) AND "R_TRIG_Sn_dx_DB".Q THEN
       "Pezzi_grigi" := "Pezzi_grigi" + 1;
   END_IF;
   IF ("Nastro_di_smistamento_sx_DB".Colore_mem = 9) AND "R_TRIG_Sn_sx_DB".Q THEN
       "Pezzi_grigi" := "Pezzi_grigi" + 1;
   END_IF;
END_REGION

REGION Network 10: Allarme Sh
   IF "Pick-place_DB".work_finished THEN "Attesa_sh" := TRUE; END_IF;
   "TON_Allarme_Sh_DB".TON(IN := "Attesa_sh" AND NOT "Sh1" AND NOT "Supervisore_DB".Cmd_Sospendi, PT := T#4s);
   IF "TON_Allarme_Sh_DB".Q THEN "Allarme_sh" := TRUE; END_IF;
   IF "Sh1" OR "Reset" OR "Supervisore_DB".Cmd_Sospendi THEN "Attesa_sh" := FALSE; END_IF;
END_REGION

REGION Network 11: Allarme colore sul nastro di smistamento destro
   IF "S_dx" THEN "Attesa_controllo_colore_dx" := TRUE; END_IF;
   "TON_Allarme_dx".TON(IN := "Attesa_controllo_colore_dx" AND ("Sc_value_dx" = 0) AND NOT "Supervisore_DB".Cmd_Sospendi,
                        PT := T#4s);
   IF "TON_Allarme_dx".Q THEN "Allarme_colore_dx" := TRUE; END_IF;
   IF ("Sc_value_dx" <> 0) OR "Reset" OR "Supervisore_DB".Cmd_Sospendi THEN
       "Attesa_controllo_colore_dx" := FALSE;
   END_IF;
END_REGION

REGION Network 12: Allarme colore sul nastro di smistamento sinistro
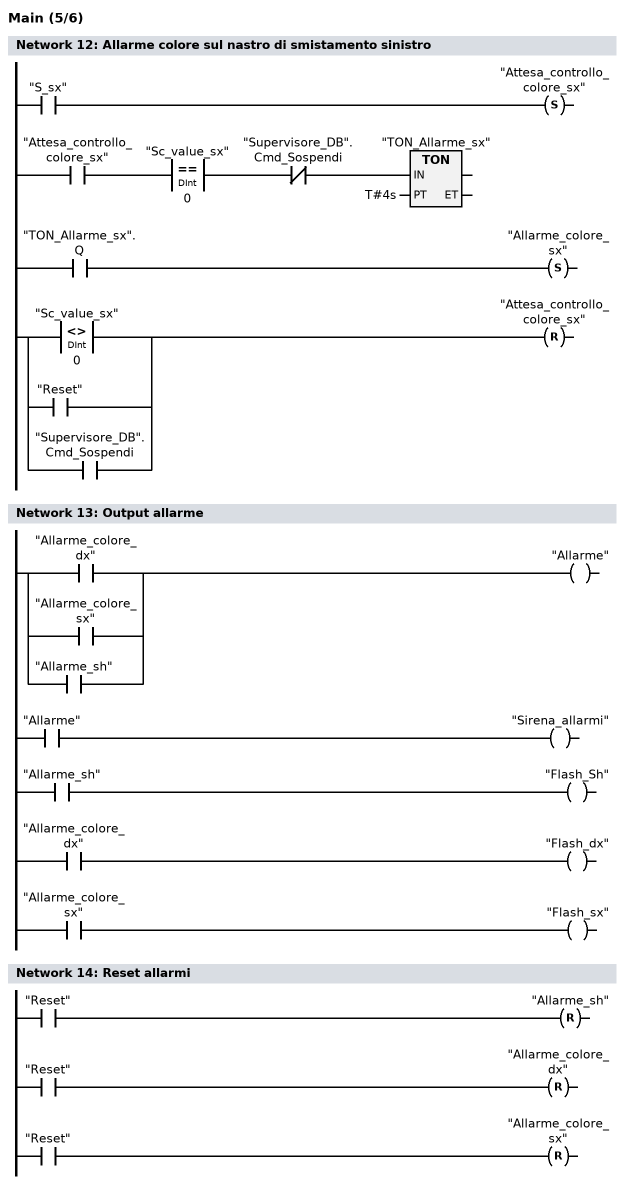
   IF "S_sx" THEN "Attesa_controllo_colore_sx" := TRUE; END_IF;
   "TON_Allarme_sx".TON(IN := "Attesa_controllo_colore_sx" AND ("Sc_value_sx" = 0) AND NOT "Supervisore_DB".Cmd_Sospendi,
                        PT := T#4s);
   IF "TON_Allarme_sx".Q THEN "Allarme_colore_sx" := TRUE; END_IF;
   IF ("Sc_value_sx" <> 0) OR "Reset" OR "Supervisore_DB".Cmd_Sospendi THEN
       "Attesa_controllo_colore_sx" := FALSE;
   END_IF;
END_REGION

REGION Network 13: Output allarme
   RUNG wire#powerrail
      Contact( "Allarme_colore_dx" )
      wire#w1
      Coil( "Allarme" )
   END_RUNG
   RUNG wire#powerrail
      Contact( "Allarme_colore_sx" )
   END_RUNG wire#w1
   RUNG wire#powerrail
      Contact( "Allarme_sh" )
   END_RUNG wire#w1
   RUNG wire#powerrail
      Contact( "Allarme" )
      Coil( "Sirena_allarmi" )
   END_RUNG
   RUNG wire#powerrail
      Contact( "Allarme_sh" )
      Coil( "Flash_Sh" )
   END_RUNG
   RUNG wire#powerrail
      Contact( "Allarme_colore_dx" )
      Coil( "Flash_dx" )
   END_RUNG
   RUNG wire#powerrail
      Contact( "Allarme_colore_sx" )
      Coil( "Flash_sx" )
   END_RUNG
   // the same network as SCL:
   "Allarme" := "Allarme_colore_dx" OR "Allarme_colore_sx" OR "Allarme_sh";
   "Sirena_allarmi" := "Allarme";
   "Flash_Sh" := "Allarme_sh";
   "Flash_dx" := "Allarme_colore_dx";
   "Flash_sx" := "Allarme_colore_sx";
END_REGION

REGION Network 14: Reset allarmi
   RUNG wire#powerrail
      Contact( "Reset" )
      R_Coil( "Allarme_sh" )
   END_RUNG
   RUNG wire#powerrail
      Contact( "Reset" )
      R_Coil( "Allarme_colore_dx" )
   END_RUNG
   RUNG wire#powerrail
      Contact( "Reset" )
      R_Coil( "Allarme_colore_sx" )
   END_RUNG
   // the same network as SCL:
   IF "Reset" THEN
       "Allarme_sh" := FALSE;
       "Allarme_colore_dx" := FALSE;
       "Allarme_colore_sx" := FALSE;
   END_IF;
END_REGION

REGION Network 15: Conversione valori allarme per allarme analogico HMI
